LIN {X 0,Y 524.503,Z 419.032,A -85,B 0,C 180,E1 -2304.785,E2 -2304.785} C_VEL
LIN {X 0,Y 515.233,Z 402.102,A -85,B 0,C 180,E1 -2307.484,E2 -2307.484} C_VEL
LIN {X 0,Y 507.271,Z 387.982,A -85,B 0,C 180,E1 -2309.916,E2 -2309.916} C_VEL
LIN {X 0,Y 504.406,Z 383.021,A -85,B 0,C 180,E1 -2310.815,E2 -2310.815} C_VEL
LIN {X 0,Y 501.74,Z 378.349,A -85,B 0,C 180,E1 -2311.688,E2 -2311.688} C_VEL
LIN {X 0,Y 499.768,Z 374.769,A -85,B 0,C 180,E1 -2312.345,E2 -2312.345} C_VEL
LIN {X 0,Y 499.108,Z 373.613,A -85,B 0,C 180,E1 -2312.564,E2 -2312.564} C_VEL
LIN {X 0,Y 497.066,Z 370.383,A -85,B 0,C 180,E1 -2313.219,E2 -2313.219} C_VEL
LIN {X 0,Y 496.734,Z 368.862,A -85,B 0,C 180,E1 -2313.458,E2 -2313.458} C_VEL
LIN {X 0,Y 496.771,Z 368.854,A -85,B 0,C 180,E1 -2317.017,E2 -2317.017} C_VEL
LIN {X 0,Y 496.751,Z 368.855,A -85,B 0,C 180,E1 -2320.481,E2 -2320.481} C_VEL
LIN {X 0,Y 496.763,Z 368.853,A -85,B 0,C 180,E1 -2323.994,E2 -2323.994} C_VEL
LIN {X 0,Y 496.722,Z 368.861,A -85,B 0,C 180,E1 -2327.562,E2 -2327.562} C_VEL
LIN {X 0,Y 496.757,Z 368.858,A -85,B 0,C 180,E1 -2331.214,E2 -2331.214} C_VEL
LIN {X 0,Y 496.754,Z 368.857,A -85,B 0,C 180,E1 -2334.688,E2 -2334.688} C_VEL
LIN {X 0,Y 496.767,Z 368.858,A -85,B 0,C 180,E1 -2338.27,E2 -2338.27} C_VEL
LIN {X 0,Y 496.741,Z 368.864,A -85,B 0,C 180,E1 -2341.73,E2 -2341.73} C_VEL
LIN {X 0,Y 496.762,Z 368.856,A -85,B 0,C 180,E1 -2345.313,E2 -2345.313} C_VEL
LIN {X 0,Y 496.739,Z 368.861,A -85,B 0,C 180,E1 -2348.772,E2 -2348.772} C_VEL
LIN {X 0,Y 496.743,Z 368.861,A -85,B 0,C 180,E1 -2352.438,E2 -2352.438} C_VEL
LIN {X 0,Y 496.77,Z 368.855,A -85,B 0,C 180,E1 -2355.887,E2 -2355.887} C_VEL
LIN {X 0,Y 496.771,Z 368.857,A -85,B 0,C 180,E1 -2359.519,E2 -2359.519} C_VEL
LIN {X 0,Y 496.746,Z 368.856,A -85,B 0,C 180,E1 -2363.095,E2 -2363.095} C_VEL
LIN {X 0,Y 496.729,Z 368.857,A -85,B 0,C 180,E1 -2366.801,E2 -2366.801} C_VEL
LIN {X 0,Y 496.772,Z 368.856,A -85,B 0,C 180,E1 -2370.344,E2 -2370.344} C_VEL
LIN {X 0,Y 496.768,Z 368.854,A -85,B 0,C 180,E1 -2373.979,E2 -2373.979} C_VEL
LIN {X 0,Y 496.751,Z 368.842,A -85,B 0,C 180,E1 -2377.53,E2 -2377.53} C_VEL
LIN {X 0,Y 496.721,Z 368.855,A -85,B 0,C 180,E1 -2381.012,E2 -2381.012} C_VEL
LIN {X 0,Y 496.77,Z 368.857,A -85,B 0,C 180,E1 -2384.462,E2 -2384.462} C_VEL
LIN {X 0,Y 496.726,Z 368.853,A -85,B 0,C 180,E1 -2387.967,E2 -2387.967} C_VEL
LIN {X 0,Y 496.762,Z 368.844,A -85,B 0,C 180,E1 -2391.542,E2 -2391.542} C_VEL
LIN {X 0,Y 496.76,Z 368.858,A -85,B 0,C 180,E1 -2392.469,E2 -2392.469} C_VEL
LIN {X 0,Y 496.68,Z 369.647,A -85,B 0,C 180,E1 -2392.956,E2 -2392.956} C_VEL
LIN {X 0,Y 496.43,Z 372.237,A -85,B 0,C 180,E1 -2393.507,E2 -2393.507} C_VEL
LIN {X 0,Y 496.098,Z 377.593,A -85,B 0,C 180,E1 -2394.159,E2 -2394.159} C_VEL
LIN {X 0,Y 496.835,Z 388.981,A -85,B 0,C 180,E1 -2395.158,E2 -2395.158} C_VEL
LIN {X 0,Y 497.729,Z 392.512,A -85,B 0,C 180,E1 -2395.508,E2 -2395.508} C_VEL
LIN {X 0,Y 500.484,Z 400.044,A -85,B 0,C 180,E1 -2396.325,E2 -2396.325} C_VEL
LIN {X 0,Y 498.752,Z 444.32,A -85,B 0,C 180,E1 -2399.73,E2 -2399.73} C_VEL
LIN {X 0,Y 497.933,Z 478.056,A -85,B 0,C 180,E1 -2402.169,E2 -2402.169} C_VEL
LIN {X 0,Y 498.047,Z 482.397,A -85,B 0,C 180,E1 -2402.43,E2 -2402.43} C_VEL
LIN {X 0,Y 499.111,Z 490.744,A -85,B 0,C 180,E1 -2402.631,E2 -2402.631} C_VEL
LIN {X 0,Y 496.753,Z 690.079,A -85,B 0,C 180,E1 -2405.69,E2 -2405.69} C_VEL
LIN {X 0,Y 496.386,Z 708.436,A -85,B 0,C 180,E1 -2406.179,E2 -2406.179} C_VEL
LIN {X 0,Y 495.792,Z 726.382,A -85,B 0,C 180,E1 -2406.87,E2 -2406.87} C_VEL
LIN {X 0,Y 495,Z 743.469,A -85,B 0,C 180,E1 -2407.745,E2 -2407.745} C_VEL
LIN {X 0,Y 494.076,Z 760.052,A -85,B 0,C 180,E1 -2408.825,E2 -2408.825} C_VEL
LIN {X 0,Y 493.114,Z 775.645,A -85,B 0,C 180,E1 -2410.084,E2 -2410.084} C_VEL
LIN {X 0,Y 492.093,Z 790.238,A -85,B 0,C 180,E1 -2411.521,E2 -2411.521} C_VEL
LIN {X 0,Y 491.127,Z 803.548,A -85,B 0,C 180,E1 -2413.108,E2 -2413.108} C_VEL
LIN {X 0,Y 490.234,Z 815.743,A -85,B 0,C 180,E1 -2414.867,E2 -2414.867} C_VEL
LIN {X 0,Y 489.489,Z 826.599,A -85,B 0,C 180,E1 -2416.775,E2 -2416.775} C_VEL
LIN {X 0,Y 488.925,Z 835.924,A -85,B 0,C 180,E1 -2418.798,E2 -2418.798} C_VEL
LIN {X 0,Y 488.507,Z 843.713,A -85,B 0,C 180,E1 -2420.933,E2 -2420.933} C_VEL
LIN {X 0,Y 488.27,Z 849.911,A -85,B 0,C 180,E1 -2423.179,E2 -2423.179} C_VEL
LIN {X 0,Y 488.161,Z 854.237,A -85,B 0,C 180,E1 -2425.419,E2 -2425.419} C_VEL
LIN {X 0,Y 488.097,Z 856.834,A -85,B 0,C 180,E1 -2427.652,E2 -2427.652} C_VEL
LIN {X 0,Y 488.082,Z 857.774,A -85,B 0,C 180,E1 -2429.883,E2 -2429.883} C_VEL
LIN {X 0,Y 488.098,Z 857.016,A -85,B 0,C 180,E1 -2432.231,E2 -2432.231} C_VEL
LIN {X 0,Y 488.156,Z 854.577,A -85,B 0,C 180,E1 -2434.464,E2 -2434.464} C_VEL
LIN {X 0,Y 488.255,Z 850.404,A -85,B 0,C 180,E1 -2436.704,E2 -2436.704} C_VEL
LIN {X 0,Y 488.47,Z 844.75,A -85,B 0,C 180,E1 -2438.831,E2 -2438.831} C_VEL
LIN {X 0,Y 488.848,Z 837.248,A -85,B 0,C 180,E1 -2440.966,E2 -2440.966} C_VEL
LIN {X 0,Y 489.381,Z 828.236,A -85,B 0,C 180,E1 -2442.988,E2 -2442.988} C_VEL
LIN {X 0,Y 490.084,Z 817.732,A -85,B 0,C 180,E1 -2444.896,E2 -2444.896} C_VEL
LIN {X 0,Y 490.962,Z 805.709,A -85,B 0,C 180,E1 -2446.688,E2 -2446.688} C_VEL
LIN {X 0,Y 491.866,Z 793.128,A -85,B 0,C 180,E1 -2448.243,E2 -2448.243} C_VEL
LIN {X 0,Y 492.899,Z 778.54,A -85,B 0,C 180,E1 -2449.739,E2 -2449.739} C_VEL
LIN {X 0,Y 493.905,Z 762.904,A -85,B 0,C 180,E1 -2451.052,E2 -2451.052} C_VEL
LIN {X 0,Y 494.82,Z 746.936,A -85,B 0,C 180,E1 -2452.139,E2 -2452.139} C_VEL
LIN {X 0,Y 495.663,Z 729.626,A -85,B 0,C 180,E1 -2453.072,E2 -2453.072} C_VEL
LIN {X 0,Y 496.319,Z 711.178,A -85,B 0,C 180,E1 -2453.824,E2 -2453.824} C_VEL
LIN {X 0,Y 496.741,Z 692.317,A -85,B 0,C 180,E1 -2454.355,E2 -2454.355} C_VEL
LIN {X 0,Y 497.123,Z 656.576,A -85,B 0,C 180,E1 -2454.939,E2 -2454.939} C_VEL
LIN {X 0,Y 498.961,Z 488.001,A -85,B 0,C 180,E1 -2457.512,E2 -2457.512} C_VEL
LIN {X 0,Y 497.92,Z 481.292,A -85,B 0,C 180,E1 -2457.702,E2 -2457.702} C_VEL
LIN {X 0,Y 498.595,Z 448.895,A -85,B 0,C 180,E1 -2460.016,E2 -2460.016} C_VEL
LIN {X 0,Y 500.418,Z 403.002,A -85,B 0,C 180,E1 -2463.543,E2 -2463.543} C_VEL
LIN {X 0,Y 500.438,Z 400,A -85,B 0,C 180,E1 -2463.782,E2 -2463.782} C_VEL
LIN {X 0,Y 492.568,Z 379.479,A -85,B 0,C 180,E1 -2466.01,E2 -2466.01} C_VEL
LIN {X 0,Y 488.944,Z 370.528,A -85,B 0,C 180,E1 -2466.986,E2 -2466.986} C_VEL
LIN {X 0,Y 488.829,Z 369.846,A -85,B 0,C 180,E1 -2467.087,E2 -2467.087} C_VEL
LIN {X 0,Y 488.778,Z 369.84,A -85,B 0,C 180,E1 -2470.449,E2 -2470.449} C_VEL
LIN {X 0,Y 488.775,Z 369.837,A -85,B 0,C 180,E1 -2474.108,E2 -2474.108} C_VEL
LIN {X 0,Y 488.822,Z 369.832,A -85,B 0,C 180,E1 -2477.596,E2 -2477.596} C_VEL
LIN {X 0,Y 488.839,Z 370.058,A -85,B 0,C 180,E1 -2479.814,E2 -2479.814} C_VEL
LIN {X 0,Y 491.722,Z 377.094,A -85,B 0,C 180,E1 -2480.78,E2 -2480.78} C_VEL
LIN {X 0,Y 500.109,Z 397.524,A -85,B 0,C 180,E1 -2483.487,E2 -2483.487} C_VEL
LIN {X 0,Y 502.886,Z 405.19,A -85,B 0,C 180,E1 -2484.432,E2 -2484.432} C_VEL
LIN {X 0,Y 500.766,Z 444.723,A -85,B 0,C 180,E1 -2487.784,E2 -2487.784} C_VEL
LIN {X 0,Y 498.572,Z 486.822,A -85,B 0,C 180,E1 -2491.294,E2 -2491.294} C_VEL
LIN {X 0,Y 496.468,Z 530.886,A -85,B 0,C 180,E1 -2494.916,E2 -2494.916} C_VEL
LIN {X 0,Y 494.54,Z 576.296,A -85,B 0,C 180,E1 -2498.596,E2 -2498.596} C_VEL
LIN {X 0,Y 493.937,Z 594.847,A -85,B 0,C 180,E1 -2500.054,E2 -2500.054} C_VEL
LIN {X 0,Y 494.638,Z 602.56,A -85,B 0,C 180,E1 -2500.224,E2 -2500.224} C_VEL
LIN {X 0,Y 492.622,Z 739.25,A -85,B 0,C 180,E1 -2502.545,E2 -2502.545} C_VEL
LIN {X 0,Y 492.328,Z 756.165,A -85,B 0,C 180,E1 -2503.063,E2 -2503.063} C_VEL
LIN {X 0,Y 491.898,Z 771.737,A -85,B 0,C 180,E1 -2503.77,E2 -2503.77} C_VEL
LIN {X 0,Y 491.359,Z 786.911,A -85,B 0,C 180,E1 -2504.697,E2 -2504.697} C_VEL
LIN {X 0,Y 490.769,Z 800.72,A -85,B 0,C 180,E1 -2505.788,E2 -2505.788} C_VEL
LIN {X 0,Y 490.179,Z 813.819,A -85,B 0,C 180,E1 -2507.093,E2 -2507.093} C_VEL
LIN {X 0,Y 489.668,Z 824.783,A -85,B 0,C 180,E1 -2508.456,E2 -2508.456} C_VEL
LIN {X 0,Y 489.189,Z 835.467,A -85,B 0,C 180,E1 -2510.121,E2 -2510.121} C_VEL
LIN {X 0,Y 488.851,Z 843.777,A -85,B 0,C 180,E1 -2511.768,E2 -2511.768} C_VEL
LIN {X 0,Y 488.601,Z 851.044,A -85,B 0,C 180,E1 -2513.655,E2 -2513.655} C_VEL
LIN {X 0,Y 488.455,Z 856.104,A -85,B 0,C 180,E1 -2515.478,E2 -2515.478} C_VEL
LIN {X 0,Y 488.405,Z 859.682,A -85,B 0,C 180,E1 -2517.484,E2 -2517.484} C_VEL
LIN {X 0,Y 488.391,Z 861.302,A -85,B 0,C 180,E1 -2519.413,E2 -2519.413} C_VEL
LIN {X 0,Y 488.438,Z 861.141,A -85,B 0,C 180,E1 -2521.407,E2 -2521.407} C_VEL
LIN {X 0,Y 488.505,Z 859.288,A -85,B 0,C 180,E1 -2523.285,E2 -2523.285} C_VEL
LIN {X 0,Y 488.672,Z 855.426,A -85,B 0,C 180,E1 -2525.283,E2 -2525.283} C_VEL
LIN {X 0,Y 488.903,Z 850.255,A -85,B 0,C 180,E1 -2527.048,E2 -2527.048} C_VEL
LIN {X 0,Y 489.295,Z 842.689,A -85,B 0,C 180,E1 -2528.934,E2 -2528.934} C_VEL
LIN {X 0,Y 489.739,Z 833.97,A -85,B 0,C 180,E1 -2530.588,E2 -2530.588} C_VEL
LIN {X 0,Y 490.294,Z 823.742,A -85,B 0,C 180,E1 -2532.125,E2 -2532.125} C_VEL
LIN {X 0,Y 490.912,Z 812.346,A -85,B 0,C 180,E1 -2533.486,E2 -2533.486} C_VEL
LIN {X 0,Y 491.551,Z 799.331,A -85,B 0,C 180,E1 -2534.729,E2 -2534.729} C_VEL
LIN {X 0,Y 492.105,Z 785.893,A -85,B 0,C 180,E1 -2535.738,E2 -2535.738} C_VEL
LIN {X 0,Y 492.623,Z 770.434,A -85,B 0,C 180,E1 -2536.629,E2 -2536.629} C_VEL
LIN {X 0,Y 492.938,Z 754.963,A -85,B 0,C 180,E1 -2537.271,E2 -2537.271} C_VEL
LIN {X 0,Y 493.11,Z 738.497,A -85,B 0,C 180,E1 -2537.722,E2 -2537.722} C_VEL
LIN {X 0,Y 495.144,Z 663.885,A -85,B 0,C 180,E1 -2539.24,E2 -2539.24} C_VEL
LIN {X 0,Y 497.519,Z 607.496,A -85,B 0,C 180,E1 -2540.468,E2 -2540.468} C_VEL
LIN {X 0,Y 498.963,Z 602.16,A -85,B 0,C 180,E1 -2540.835,E2 -2540.835} C_VEL
LIN {X 0,Y 502.913,Z 561.509,A -85,B 0,C 180,E1 -2544.489,E2 -2544.489} C_VEL
LIN {X 0,Y 508.091,Z 522.478,A -85,B 0,C 180,E1 -2548.183,E2 -2548.183} C_VEL
LIN {X 0,Y 513.352,Z 494.26,A -85,B 0,C 180,E1 -2551.019,E2 -2551.019} C_VEL
LIN {X 0,Y 519.178,Z 471.939,A -85,B 0,C 180,E1 -2553.421,E2 -2553.421} C_VEL
LIN {X 0,Y 525.35,Z 455.383,A -85,B 0,C 180,E1 -2555.35,E2 -2555.35} C_VEL
LIN {X 0,Y 527.979,Z 449.901,A -85,B 0,C 180,E1 -2556.037,E2 -2556.037} C_VEL
LIN {X 0,Y 520.798,Z 461.366,A -85,B 0,C 180,E1 -2557.27,E2 -2557.27} C_VEL
LIN {X 0,Y 516.041,Z 472.438,A -85,B 0,C 180,E1 -2558.484,E2 -2558.484} C_VEL
LIN {X 0,Y 513.414,Z 483.465,A -85,B 0,C 180,E1 -2559.713,E2 -2559.713} C_VEL
LIN {X 0,Y 512.933,Z 495.108,A -85,B 0,C 180,E1 -2561.028,E2 -2561.028} C_VEL
LIN {X 0,Y 514.549,Z 505.694,A -85,B 0,C 180,E1 -2562.247,E2 -2562.247} C_VEL
LIN {X 0,Y 518.036,Z 515.468,A -85,B 0,C 180,E1 -2563.402,E2 -2563.402} C_VEL
LIN {X 0,Y 523.717,Z 525.213,A -85,B 0,C 180,E1 -2564.592,E2 -2564.592} C_VEL
LIN {X 0,Y 531.685,Z 534.476,A -85,B 0,C 180,E1 -2565.765,E2 -2565.765} C_VEL
LIN {X 0,Y 541.467,Z 542.475,A -85,B 0,C 180,E1 -2566.835,E2 -2566.835} C_VEL
LIN {X 0,Y 552.276,Z 548.88,A -85,B 0,C 180,E1 -2567.771,E2 -2567.771} C_VEL
LIN {X 0,Y 562.809,Z 553.266,A -85,B 0,C 180,E1 -2568.564,E2 -2568.564} C_VEL
LIN {X 0,Y 567.662,Z 554.303,A -85,B 0,C 180,E1 -2569.08,E2 -2569.08} C_VEL
LIN {X 0,Y 570.982,Z 554.208,A -85,B 0,C 180,E1 -2569.617,E2 -2569.617} C_VEL
LIN {X 0,Y 573.098,Z 553.255,A -85,B 0,C 180,E1 -2570.186,E2 -2570.186} C_VEL
LIN {X 0,Y 573.653,Z 552.573,A -85,B 0,C 180,E1 -2570.46,E2 -2570.46} C_VEL
LIN {X 0,Y 566.628,Z 573.364,A -85,B 0,C 180,E1 -2570.751,E2 -2570.751} C_VEL
LIN {X 0,Y 562.375,Z 585.951,A -85,B 0,C 180,E1 -2571.06,E2 -2571.06} C_VEL
LIN {X 0,Y 553.254,Z 606.117,A -85,B 0,C 180,E1 -2571.202,E2 -2571.202} C_VEL
LIN {X 0,Y 542.151,Z 627.242,A -85,B 0,C 180,E1 -2571.506,E2 -2571.506} C_VEL
LIN {X 0,Y 532.299,Z 645.678,A -85,B 0,C 180,E1 -2571.967,E2 -2571.967} C_VEL
LIN {X 0,Y 525.341,Z 661.055,A -85,B 0,C 180,E1 -2572.479,E2 -2572.479} C_VEL
LIN {X 0,Y 521.674,Z 671.361,A -85,B 0,C 180,E1 -2572.874,E2 -2572.874} C_VEL
LIN {X 0,Y 515.253,Z 685.606,A -85,B 0,C 180,E1 -2573.365,E2 -2573.365} C_VEL
LIN {X 0,Y 507.043,Z 711.323,A -85,B 0,C 180,E1 -2574.428,E2 -2574.428} C_VEL
LIN {X 0,Y 504.91,Z 720.444,A -85,B 0,C 180,E1 -2574.812,E2 -2574.812} C_VEL
LIN {X 0,Y 504.327,Z 762.509,A -85,B 0,C 180,E1 -2575.46,E2 -2575.46} C_VEL
LIN {X 0,Y 503.48,Z 786.582,A -85,B 0,C 180,E1 -2576.043,E2 -2576.043} C_VEL
LIN {X 0,Y 502.543,Z 808.772,A -85,B 0,C 180,E1 -2576.794,E2 -2576.794} C_VEL
LIN {X 0,Y 501.448,Z 827.405,A -85,B 0,C 180,E1 -2577.63,E2 -2577.63} C_VEL
LIN {X 0,Y 499.915,Z 846.819,A -85,B 0,C 180,E1 -2578.733,E2 -2578.733} C_VEL
LIN {X 0,Y 498.233,Z 866.627,A -85,B 0,C 180,E1 -2580.104,E2 -2580.104} C_VEL
LIN {X 0,Y 496.476,Z 885.398,A -85,B 0,C 180,E1 -2581.651,E2 -2581.651} C_VEL
LIN {X 0,Y 494.727,Z 904.088,A -85,B 0,C 180,E1 -2583.471,E2 -2583.471} C_VEL
LIN {X 0,Y 493.156,Z 920.729,A -85,B 0,C 180,E1 -2585.377,E2 -2585.377} C_VEL
LIN {X 0,Y 491.772,Z 935.909,A -85,B 0,C 180,E1 -2587.401,E2 -2587.401} C_VEL
LIN {X 0,Y 490.566,Z 950.305,A -85,B 0,C 180,E1 -2589.645,E2 -2589.645} C_VEL
LIN {X 0,Y 489.601,Z 963.337,A -85,B 0,C 180,E1 -2592.039,E2 -2592.039} C_VEL
LIN {X 0,Y 488.902,Z 974.404,A -85,B 0,C 180,E1 -2594.46,E2 -2594.46} C_VEL
LIN {X 0,Y 488.404,Z 984.338,A -85,B 0,C 180,E1 -2597.106,E2 -2597.106} C_VEL
LIN {X 0,Y 488.115,Z 992.2,A -85,B 0,C 180,E1 -2599.734,E2 -2599.734} C_VEL
LIN {X 0,Y 487.964,Z 998.151,A -85,B 0,C 180,E1 -2602.346,E2 -2602.346} C_VEL
LIN {X 0,Y 487.907,Z 1002.147,A -85,B 0,C 180,E1 -2604.838,E2 -2604.838} C_VEL
LIN {X 0,Y 487.895,Z 1004.524,A -85,B 0,C 180,E1 -2607.298,E2 -2607.298} C_VEL
LIN {X 0,Y 487.897,Z 1005.44,A -85,B 0,C 180,E1 -2609.647,E2 -2609.647} C_VEL
LIN {X 0,Y 487.91,Z 1004.912,A -85,B 0,C 180,E1 -2612.114,E2 -2612.114} C_VEL
LIN {X 0,Y 487.912,Z 1002.74,A -85,B 0,C 180,E1 -2614.702,E2 -2614.702} C_VEL
LIN {X 0,Y 487.947,Z 998.808,A -85,B 0,C 180,E1 -2617.299,E2 -2617.299} C_VEL
LIN {X 0,Y 488.067,Z 993.353,A -85,B 0,C 180,E1 -2619.811,E2 -2619.811} C_VEL
LIN {X 0,Y 488.311,Z 986.309,A -85,B 0,C 180,E1 -2622.295,E2 -2622.295} C_VEL
LIN {X 0,Y 488.737,Z 977.337,A -85,B 0,C 180,E1 -2624.816,E2 -2624.816} C_VEL
LIN {X 0,Y 489.401,Z 966.295,A -85,B 0,C 180,E1 -2627.354,E2 -2627.354} C_VEL
LIN {X 0,Y 490.31,Z 953.621,A -85,B 0,C 180,E1 -2629.786,E2 -2629.786} C_VEL
LIN {X 0,Y 491.493,Z 939.294,A -85,B 0,C 180,E1 -2632.108,E2 -2632.108} C_VEL
LIN {X 0,Y 492.935,Z 923.225,A -85,B 0,C 180,E1 -2634.315,E2 -2634.315} C_VEL
LIN {X 0,Y 494.614,Z 905.274,A -85,B 0,C 180,E1 -2636.406,E2 -2636.406} C_VEL
LIN {X 0,Y 496.38,Z 886.455,A -85,B 0,C 180,E1 -2638.252,E2 -2638.252} C_VEL
LIN {X 0,Y 498.176,Z 867.207,A -85,B 0,C 180,E1 -2639.851,E2 -2639.851} C_VEL
LIN {X 0,Y 499.838,Z 847.827,A -85,B 0,C 180,E1 -2641.204,E2 -2641.204} C_VEL
LIN {X 0,Y 501.365,Z 828.672,A -85,B 0,C 180,E1 -2642.307,E2 -2642.307} C_VEL
LIN {X 0,Y 502.601,Z 808.206,A -85,B 0,C 180,E1 -2643.234,E2 -2643.234} C_VEL
LIN {X 0,Y 503.712,Z 785.487,A -85,B 0,C 180,E1 -2644.029,E2 -2644.029} C_VEL
LIN {X 0,Y 504.625,Z 762.44,A -85,B 0,C 180,E1 -2644.609,E2 -2644.609} C_VEL
LIN {X 0,Y 505.297,Z 722.062,A -85,B 0,C 180,E1 -2645.262,E2 -2645.262} C_VEL
LIN {X 0,Y 505.606,Z 719.266,A -85,B 0,C 180,E1 -2645.34,E2 -2645.34} C_VEL
LIN {X 0,Y 509.96,Z 703.556,A -85,B 0,C 180,E1 -2646.029,E2 -2646.029} C_VEL
LIN {X 0,Y 516.417,Z 684.139,A -85,B 0,C 180,E1 -2646.795,E2 -2646.795} C_VEL
LIN {X 0,Y 522.774,Z 669.701,A -85,B 0,C 180,E1 -2647.253,E2 -2647.253} C_VEL
LIN {X 0,Y 527.202,Z 657.309,A -85,B 0,C 180,E1 -2647.707,E2 -2647.707} C_VEL
LIN {X 0,Y 535.529,Z 639.572,A -85,B 0,C 180,E1 -2648.214,E2 -2648.214} C_VEL
LIN {X 0,Y 546.551,Z 619.139,A -85,B 0,C 180,E1 -2648.634,E2 -2648.634} C_VEL
LIN {X 0,Y 556.954,Z 598.362,A -85,B 0,C 180,E1 -2648.867,E2 -2648.867} C_VEL
LIN {X 0,Y 562.84,Z 584.646,A -85,B 0,C 180,E1 -2648.966,E2 -2648.966} C_VEL
LIN {X 0,Y 567.532,Z 570.757,A -85,B 0,C 180,E1 -2649.298,E2 -2649.298} C_VEL
LIN {X 0,Y 573.649,Z 552.565,A -85,B 0,C 180,E1 -2649.551,E2 -2649.551} C_VEL
LIN {X 0,Y 571.887,Z 553.958,A -85,B 0,C 180,E1 -2650.18,E2 -2650.18} C_VEL
LIN {X 0,Y 568.861,Z 554.372,A -85,B 0,C 180,E1 -2650.752,E2 -2650.752} C_VEL
LIN {X 0,Y 565.013,Z 553.856,A -85,B 0,C 180,E1 -2651.229,E2 -2651.229} C_VEL
LIN {X 0,Y 554.055,Z 550.104,A -85,B 0,C 180,E1 -2652.308,E2 -2652.308} C_VEL
LIN {X 0,Y 544.18,Z 544.7,A -85,B 0,C 180,E1 -2653.468,E2 -2653.468} C_VEL
LIN {X 0,Y 535.663,Z 537.821,A -85,B 0,C 180,E1 -2654.67,E2 -2654.67} C_VEL
LIN {X 0,Y 528.131,Z 528.834,A -85,B 0,C 180,E1 -2655.989,E2 -2655.989} C_VEL
LIN {X 0,Y 522.652,Z 519.047,A -85,B 0,C 180,E1 -2657.225,E2 -2657.225} C_VEL
LIN {X 0,Y 518.636,Z 507.922,A -85,B 0,C 180,E1 -2658.457,E2 -2658.457} C_VEL
LIN {X 0,Y 516.125,Z 495.378,A -85,B 0,C 180,E1 -2659.682,E2 -2659.682} C_VEL
LIN {X 0,Y 514.966,Z 479.928,A -85,B 0,C 180,E1 -2661.018,E2 -2661.018} C_VEL
LIN {X 0,Y 515.59,Z 460.544,A -85,B 0,C 180,E1 -2662.489,E2 -2662.489} C_VEL
LIN {X 0,Y 518.516,Z 423.387,A -85,B 0,C 180,E1 -2665.196,E2 -2665.196} C_VEL
LIN {X 0,Y 509.071,Z 406.235,A -85,B 0,C 180,E1 -2667.974,E2 -2667.974} C_VEL
LIN {X 0,Y 502.092,Z 393.774,A -85,B 0,C 180,E1 -2670.143,E2 -2670.143} C_VEL
LIN {X 0,Y 496.676,Z 384.303,A -85,B 0,C 180,E1 -2671.897,E2 -2671.897} C_VEL
LIN {X 0,Y 494.04,Z 379.628,A -85,B 0,C 180,E1 -2672.782,E2 -2672.782} C_VEL
LIN {X 0,Y 492.051,Z 376.345,A -85,B 0,C 180,E1 -2673.446,E2 -2673.446} C_VEL
LIN {X 0,Y 491.125,Z 374.539,A -85,B 0,C 180,E1 -2673.783,E2 -2673.783} C_VEL
LIN {X 0,Y 489.128,Z 371.287,A -85,B 0,C 180,E1 -2674.449,E2 -2674.449} C_VEL
LIN {X 0,Y 488.803,Z 369.847,A -85,B 0,C 180,E1 -2674.705,E2 -2674.705} C_VEL
LIN {X 0,Y 488.835,Z 369.843,A -85,B 0,C 180,E1 -2678.271,E2 -2678.271} C_VEL
LIN {X 0,Y 488.828,Z 369.843,A -85,B 0,C 180,E1 -2682.011,E2 -2682.011} C_VEL
LIN {X 0,Y 488.809,Z 369.847,A -85,B 0,C 180,E1 -2685.549,E2 -2685.549} C_VEL
LIN {X 0,Y 488.796,Z 369.849,A -85,B 0,C 180,E1 -2689.153,E2 -2689.153} C_VEL
LIN {X 0,Y 488.828,Z 369.844,A -85,B 0,C 180,E1 -2692.597,E2 -2692.597} C_VEL
LIN {X 0,Y 488.798,Z 369.849,A -85,B 0,C 180,E1 -2696.247,E2 -2696.247} C_VEL
LIN {X 0,Y 488.832,Z 369.85,A -85,B 0,C 180,E1 -2699.766,E2 -2699.766} C_VEL
LIN {X 0,Y 488.81,Z 369.851,A -85,B 0,C 180,E1 -2703.284,E2 -2703.284} C_VEL
LIN {X 0,Y 488.823,Z 369.848,A -85,B 0,C 180,E1 -2706.814,E2 -2706.814} C_VEL
LIN {X 0,Y 488.781,Z 369.848,A -85,B 0,C 180,E1 -2710.371,E2 -2710.371} C_VEL
LIN {X 0,Y 488.821,Z 369.846,A -85,B 0,C 180,E1 -2713.967,E2 -2713.967} C_VEL
LIN {X 0,Y 488.818,Z 369.848,A -85,B 0,C 180,E1 -2717.499,E2 -2717.499} C_VEL
LIN {X 0,Y 488.829,Z 369.844,A -85,B 0,C 180,E1 -2721.1,E2 -2721.1} C_VEL
LIN {X 0,Y 488.789,Z 369.849,A -85,B 0,C 180,E1 -2724.665,E2 -2724.665} C_VEL
LIN {X 0,Y 488.816,Z 369.842,A -85,B 0,C 180,E1 -2728.33,E2 -2728.33} C_VEL
LIN {X 0,Y 488.805,Z 369.84,A -85,B 0,C 180,E1 -2731.716,E2 -2731.716} C_VEL
LIN {X 0,Y 488.812,Z 369.831,A -85,B 0,C 180,E1 -2735.299,E2 -2735.299} C_VEL
LIN {X 0,Y 488.826,Z 369.843,A -85,B 0,C 180,E1 -2738.803,E2 -2738.803} C_VEL
LIN {X 0,Y 488.824,Z 369.826,A -85,B 0,C 180,E1 -2742.454,E2 -2742.454} C_VEL
LIN {X 0,Y 488.804,Z 369.845,A -85,B 0,C 180,E1 -2745.935,E2 -2745.935} C_VEL
LIN {X 0,Y 488.795,Z 369.854,A -85,B 0,C 180,E1 -2749.576,E2 -2749.576} C_VEL
LIN {X 0,Y 488.855,Z 370.012,A -85,B 0,C 180,E1 -2753.062,E2 -2753.062} C_VEL
LIN {X 0,Y 497.729,Z 392.512,A -85,B 0,C 180,E1 -2755.508,E2 -2755.508} C_VEL
LIN {X 0,Y 498.073,Z 395.994,A -85,B 0,C 180,E1 -2755.811,E2 -2755.811} C_VEL
LIN {X 0,Y 496.56,Z 401.823,A -85,B 0,C 180,E1 -2756.156,E2 -2756.156} C_VEL
LIN {X 0,Y 493.439,Z 410.585,A -85,B 0,C 180,E1 -2756.62,E2 -2756.62} C_VEL
LIN {X 0,Y 493.054,Z 413.215,A -85,B 0,C 180,E1 -2756.804,E2 -2756.804} C_VEL
LIN {X 0,Y 491.393,Z 456.207,A -85,B 0,C 180,E1 -2760.099,E2 -2760.099} C_VEL
LIN {X 0,Y 490.934,Z 483.139,A -85,B 0,C 180,E1 -2761.989,E2 -2761.989} C_VEL
LIN {X 0,Y 492.064,Z 491.769,A -85,B 0,C 180,E1 -2762.204,E2 -2762.204} C_VEL
LIN {X 0,Y 489.525,Z 691.201,A -85,B 0,C 180,E1 -2765.307,E2 -2765.307} C_VEL
LIN {X 0,Y 489.144,Z 709.676,A -85,B 0,C 180,E1 -2765.805,E2 -2765.805} C_VEL
LIN {X 0,Y 488.522,Z 727.692,A -85,B 0,C 180,E1 -2766.51,E2 -2766.51} C_VEL
LIN {X 0,Y 487.691,Z 744.691,A -85,B 0,C 180,E1 -2767.393,E2 -2767.393} C_VEL
LIN {X 0,Y 486.71,Z 761.37,A -85,B 0,C 180,E1 -2768.495,E2 -2768.495} C_VEL
LIN {X 0,Y 485.688,Z 776.887,A -85,B 0,C 180,E1 -2769.767,E2 -2769.767} C_VEL
LIN {X 0,Y 484.595,Z 791.488,A -85,B 0,C 180,E1 -2771.224,E2 -2771.224} C_VEL
LIN {X 0,Y 483.576,Z 804.561,A -85,B 0,C 180,E1 -2772.803,E2 -2772.803} C_VEL
LIN {X 0,Y 482.592,Z 817.003,A -85,B 0,C 180,E1 -2774.622,E2 -2774.622} C_VEL
LIN {X 0,Y 481.778,Z 827.862,A -85,B 0,C 180,E1 -2776.56,E2 -2776.56} C_VEL
LIN {X 0,Y 481.153,Z 837.189,A -85,B 0,C 180,E1 -2778.615,E2 -2778.615} C_VEL
LIN {X 0,Y 480.685,Z 844.979,A -85,B 0,C 180,E1 -2780.784,E2 -2780.784} C_VEL
LIN {X 0,Y 480.411,Z 851.177,A -85,B 0,C 180,E1 -2783.067,E2 -2783.067} C_VEL
LIN {X 0,Y 480.278,Z 855.502,A -85,B 0,C 180,E1 -2785.343,E2 -2785.343} C_VEL
LIN {X 0,Y 480.202,Z 858.098,A -85,B 0,C 180,E1 -2787.614,E2 -2787.614} C_VEL
LIN {X 0,Y 480.183,Z 859.038,A -85,B 0,C 180,E1 -2789.881,E2 -2789.881} C_VEL
LIN {X 0,Y 480.202,Z 858.279,A -85,B 0,C 180,E1 -2792.268,E2 -2792.268} C_VEL
LIN {X 0,Y 480.273,Z 855.839,A -85,B 0,C 180,E1 -2794.538,E2 -2794.538} C_VEL
LIN {X 0,Y 480.394,Z 851.667,A -85,B 0,C 180,E1 -2796.814,E2 -2796.814} C_VEL
LIN {X 0,Y 480.642,Z 846.011,A -85,B 0,C 180,E1 -2798.976,E2 -2798.976} C_VEL
LIN {X 0,Y 481.068,Z 838.508,A -85,B 0,C 180,E1 -2801.145,E2 -2801.145} C_VEL
LIN {X 0,Y 481.659,Z 829.493,A -85,B 0,C 180,E1 -2803.2,E2 -2803.2} C_VEL
LIN {X 0,Y 482.429,Z 818.984,A -85,B 0,C 180,E1 -2805.138,E2 -2805.138} C_VEL
LIN {X 0,Y 483.379,Z 806.955,A -85,B 0,C 180,E1 -2806.957,E2 -2806.957} C_VEL
LIN {X 0,Y 484.397,Z 793.84,A -85,B 0,C 180,E1 -2808.597,E2 -2808.597} C_VEL
LIN {X 0,Y 485.495,Z 779.333,A -85,B 0,C 180,E1 -2810.096,E2 -2810.096} C_VEL
LIN {X 0,Y 486.566,Z 763.623,A -85,B 0,C 180,E1 -2811.426,E2 -2811.426} C_VEL
LIN {X 0,Y 487.562,Z 747.183,A -85,B 0,C 180,E1 -2812.55,E2 -2812.55} C_VEL
LIN {X 0,Y 488.462,Z 729.443,A -85,B 0,C 180,E1 -2813.503,E2 -2813.503} C_VEL
LIN {X 0,Y 489.112,Z 710.984,A -85,B 0,C 180,E1 -2814.243,E2 -2814.243} C_VEL
LIN {X 0,Y 489.518,Z 692.403,A -85,B 0,C 180,E1 -2814.758,E2 -2814.758} C_VEL
LIN {X 0,Y 490.104,Z 642.033,A -85,B 0,C 180,E1 -2815.57,E2 -2815.57} C_VEL
LIN {X 0,Y 491.911,Z 489.03,A -85,B 0,C 180,E1 -2817.942,E2 -2817.942} C_VEL
LIN {X 0,Y 490.878,Z 482.661,A -85,B 0,C 180,E1 -2818.119,E2 -2818.119} C_VEL
LIN {X 0,Y 491.556,Z 450.643,A -85,B 0,C 180,E1 -2820.407,E2 -2820.407} C_VEL
LIN {X 0,Y 493.432,Z 404.906,A -85,B 0,C 180,E1 -2823.936,E2 -2823.936} C_VEL
LIN {X 0,Y 493.32,Z 402.834,A -85,B 0,C 180,E1 -2824.111,E2 -2824.111} C_VEL
LIN {X 0,Y 485.048,Z 381.238,A -85,B 0,C 180,E1 -2826.492,E2 -2826.492} C_VEL
LIN {X 0,Y 480.904,Z 371.185,A -85,B 0,C 180,E1 -2827.613,E2 -2827.613} C_VEL
LIN {X 0,Y 480.849,Z 370.84,A -85,B 0,C 180,E1 -2827.686,E2 -2827.686} C_VEL
LIN {X 0,Y 480.899,Z 370.822,A -85,B 0,C 180,E1 -2831.179,E2 -2831.179} C_VEL
LIN {X 0,Y 480.842,Z 370.823,A -85,B 0,C 180,E1 -2834.671,E2 -2834.671} C_VEL
LIN {X 0,Y 480.837,Z 370.825,A -85,B 0,C 180,E1 -2838.29,E2 -2838.29} C_VEL
LIN {X 0,Y 480.888,Z 371.027,A -85,B 0,C 180,E1 -2839.084,E2 -2839.084} C_VEL
LIN {X 0,Y 490.099,Z 393.057,A -85,B 0,C 180,E1 -2842.142,E2 -2842.142} C_VEL
LIN {X 0,Y 496.011,Z 408.442,A -85,B 0,C 180,E1 -2844.116,E2 -2844.116} C_VEL
LIN {X 0,Y 493.608,Z 449.502,A -85,B 0,C 180,E1 -2847.638,E2 -2847.638} C_VEL
LIN {X 0,Y 491.327,Z 491.53,A -85,B 0,C 180,E1 -2851.164,E2 -2851.164} C_VEL
LIN {X 0,Y 489.044,Z 536.834,A -85,B 0,C 180,E1 -2854.922,E2 -2854.922} C_VEL
LIN {X 0,Y 486.925,Z 584.474,A -85,B 0,C 180,E1 -2858.813,E2 -2858.813} C_VEL
LIN {X 0,Y 486.56,Z 595.568,A -85,B 0,C 180,E1 -2859.683,E2 -2859.683} C_VEL
LIN {X 0,Y 487.281,Z 603.269,A -85,B 0,C 180,E1 -2859.864,E2 -2859.864} C_VEL
LIN {X 0,Y 485.047,Z 740.362,A -85,B 0,C 180,E1 -2862.261,E2 -2862.261} C_VEL
LIN {X 0,Y 484.734,Z 757.33,A -85,B 0,C 180,E1 -2862.793,E2 -2862.793} C_VEL
LIN {X 0,Y 484.281,Z 772.764,A -85,B 0,C 180,E1 -2863.507,E2 -2863.507} C_VEL
LIN {X 0,Y 483.699,Z 788.281,A -85,B 0,C 180,E1 -2864.473,E2 -2864.473} C_VEL
LIN {X 0,Y 483.084,Z 801.761,A -85,B 0,C 180,E1 -2865.557,E2 -2865.557} C_VEL
LIN {X 0,Y 482.477,Z 814.336,A -85,B 0,C 180,E1 -2866.823,E2 -2866.823} C_VEL
LIN {X 0,Y 481.902,Z 825.882,A -85,B 0,C 180,E1 -2868.268,E2 -2868.268} C_VEL
LIN {X 0,Y 481.385,Z 836.563,A -85,B 0,C 180,E1 -2869.952,E2 -2869.952} C_VEL
LIN {X 0,Y 481.014,Z 844.956,A -85,B 0,C 180,E1 -2871.633,E2 -2871.633} C_VEL
LIN {X 0,Y 480.739,Z 852.269,A -85,B 0,C 180,E1 -2873.551,E2 -2873.551} C_VEL
LIN {X 0,Y 480.583,Z 857.245,A -85,B 0,C 180,E1 -2875.346,E2 -2875.346} C_VEL
LIN {X 0,Y 480.521,Z 860.901,A -85,B 0,C 180,E1 -2877.376,E2 -2877.376} C_VEL
LIN {X 0,Y 480.508,Z 862.618,A -85,B 0,C 180,E1 -2879.284,E2 -2879.284} C_VEL
LIN {X 0,Y 480.556,Z 862.581,A -85,B 0,C 180,E1 -2881.311,E2 -2881.311} C_VEL
LIN {X 0,Y 480.641,Z 860.886,A -85,B 0,C 180,E1 -2883.219,E2 -2883.219} C_VEL
LIN {X 0,Y 480.82,Z 857.15,A -85,B 0,C 180,E1 -2885.249,E2 -2885.249} C_VEL
LIN {X 0,Y 481.082,Z 852.153,A -85,B 0,C 180,E1 -2887.043,E2 -2887.043} C_VEL
LIN {X 0,Y 481.464,Z 845.251,A -85,B 0,C 180,E1 -2888.84,E2 -2888.84} C_VEL
LIN {X 0,Y 481.956,Z 836.932,A -85,B 0,C 180,E1 -2890.519,E2 -2890.519} C_VEL
LIN {X 0,Y 482.525,Z 827.033,A -85,B 0,C 180,E1 -2892.08,E2 -2892.08} C_VEL
LIN {X 0,Y 483.204,Z 815.648,A -85,B 0,C 180,E1 -2893.522,E2 -2893.522} C_VEL
LIN {X 0,Y 483.875,Z 803.132,A -85,B 0,C 180,E1 -2894.779,E2 -2894.779} C_VEL
LIN {X 0,Y 484.522,Z 789.543,A -85,B 0,C 180,E1 -2895.868,E2 -2895.868} C_VEL
LIN {X 0,Y 485.042,Z 774.737,A -85,B 0,C 180,E1 -2896.773,E2 -2896.773} C_VEL
LIN {X 0,Y 485.439,Z 759.257,A -85,B 0,C 180,E1 -2897.477,E2 -2897.477} C_VEL
LIN {X 0,Y 485.626,Z 742.723,A -85,B 0,C 180,E1 -2897.973,E2 -2897.973} C_VEL
LIN {X 0,Y 487.821,Z 670.656,A -85,B 0,C 180,E1 -2899.533,E2 -2899.533} C_VEL
LIN {X 0,Y 490.82,Z 609.716,A -85,B 0,C 180,E1 -2900.947,E2 -2900.947} C_VEL
LIN {X 0,Y 492.502,Z 603.638,A -85,B 0,C 180,E1 -2901.371,E2 -2901.371} C_VEL
LIN {X 0,Y 497.184,Z 560.839,A -85,B 0,C 180,E1 -2905.299,E2 -2905.299} C_VEL
LIN {X 0,Y 502.752,Z 523.775,A -85,B 0,C 180,E1 -2908.899,E2 -2908.899} C_VEL
LIN {X 0,Y 508.269,Z 497.727,A -85,B 0,C 180,E1 -2911.592,E2 -2911.592} C_VEL
LIN {X 0,Y 514.093,Z 477.831,A -85,B 0,C 180,E1 -2913.796,E2 -2913.796} C_VEL
LIN {X 0,Y 520.513,Z 462.288,A -85,B 0,C 180,E1 -2915.654,E2 -2915.654} C_VEL
LIN {X 0,Y 521.646,Z 460.023,A -85,B 0,C 180,E1 -2915.968,E2 -2915.968} C_VEL
LIN {X 0,Y 514.762,Z 471.03,A -85,B 0,C 180,E1 -2917.214,E2 -2917.214} C_VEL
LIN {X 0,Y 510.208,Z 481.828,A -85,B 0,C 180,E1 -2918.472,E2 -2918.472} C_VEL
LIN {X 0,Y 507.95,Z 491.919,A -85,B 0,C 180,E1 -2919.677,E2 -2919.677} C_VEL
LIN {X 0,Y 507.649,Z 502.763,A -85,B 0,C 180,E1 -2920.985,E2 -2920.985} C_VEL
LIN {X 0,Y 509.591,Z 513.482,A -85,B 0,C 180,E1 -2922.298,E2 -2922.298} C_VEL
LIN {X 0,Y 513.205,Z 522.69,A -85,B 0,C 180,E1 -2923.451,E2 -2923.451} C_VEL
LIN {X 0,Y 518.563,Z 531.482,A -85,B 0,C 180,E1 -2924.574,E2 -2924.574} C_VEL
LIN {X 0,Y 526.289,Z 540.379,A -85,B 0,C 180,E1 -2925.744,E2 -2925.744} C_VEL
LIN {X 0,Y 535.951,Z 548.334,A -85,B 0,C 180,E1 -2926.839,E2 -2926.839} C_VEL
LIN {X 0,Y 547.472,Z 555.259,A -85,B 0,C 180,E1 -2927.858,E2 -2927.858} C_VEL
LIN {X 0,Y 559.715,Z 560.386,A -85,B 0,C 180,E1 -2928.769,E2 -2928.769} C_VEL
LIN {X 0,Y 564.758,Z 561.529,A -85,B 0,C 180,E1 -2929.265,E2 -2929.265} C_VEL
LIN {X 0,Y 568.232,Z 561.713,A -85,B 0,C 180,E1 -2929.798,E2 -2929.798} C_VEL
LIN {X 0,Y 561.005,Z 579.487,A -85,B 0,C 180,E1 -2930.154,E2 -2930.154} C_VEL
LIN {X 0,Y 558.539,Z 586.008,A -85,B 0,C 180,E1 -2930.332,E2 -2930.332} C_VEL
LIN {X 0,Y 547.964,Z 605.065,A -85,B 0,C 180,E1 -2930.58,E2 -2930.58} C_VEL
LIN {X 0,Y 533.173,Z 629.737,A -85,B 0,C 180,E1 -2931.149,E2 -2931.149} C_VEL
LIN {X 0,Y 522.892,Z 649.225,A -85,B 0,C 180,E1 -2931.717,E2 -2931.717} C_VEL
LIN {X 0,Y 516.784,Z 663.945,A -85,B 0,C 180,E1 -2932.24,E2 -2932.24} C_VEL
LIN {X 0,Y 514.597,Z 670.004,A -85,B 0,C 180,E1 -2932.473,E2 -2932.473} C_VEL
LIN {X 0,Y 508.121,Z 684.48,A -85,B 0,C 180,E1 -2932.977,E2 -2932.977} C_VEL
LIN {X 0,Y 499.836,Z 710.258,A -85,B 0,C 180,E1 -2934.047,E2 -2934.047} C_VEL
LIN {X 0,Y 497.751,Z 718.943,A -85,B 0,C 180,E1 -2934.415,E2 -2934.415} C_VEL
LIN {X 0,Y 496.996,Z 761.232,A -85,B 0,C 180,E1 -2935.076,E2 -2935.076} C_VEL
LIN {X 0,Y 496.1,Z 785.159,A -85,B 0,C 180,E1 -2935.664,E2 -2935.664} C_VEL
LIN {X 0,Y 495.065,Z 807.747,A -85,B 0,C 180,E1 -2936.435,E2 -2936.435} C_VEL
LIN {X 0,Y 493.81,Z 829.795,A -85,B 0,C 180,E1 -2937.412,E2 -2937.412} C_VEL
LIN {X 0,Y 492.4,Z 850.479,A -85,B 0,C 180,E1 -2938.542,E2 -2938.542} C_VEL
LIN {X 0,Y 491.075,Z 867.33,A -85,B 0,C 180,E1 -2939.687,E2 -2939.687} C_VEL
LIN {X 0,Y 489.302,Z 885.09,A -85,B 0,C 180,E1 -2941.167,E2 -2941.167} C_VEL
LIN {X 0,Y 487.436,Z 903.498,A -85,B 0,C 180,E1 -2942.976,E2 -2942.976} C_VEL
LIN {X 0,Y 485.711,Z 920.23,A -85,B 0,C 180,E1 -2944.908,E2 -2944.908} C_VEL
LIN {X 0,Y 484.158,Z 935.911,A -85,B 0,C 180,E1 -2947.026,E2 -2947.026} C_VEL
LIN {X 0,Y 482.865,Z 950.066,A -85,B 0,C 180,E1 -2949.262,E2 -2949.262} C_VEL
LIN {X 0,Y 481.83,Z 962.743,A -85,B 0,C 180,E1 -2951.613,E2 -2951.613} C_VEL
LIN {X 0,Y 480.999,Z 974.607,A -85,B 0,C 180,E1 -2954.246,E2 -2954.246} C_VEL
LIN {X 0,Y 480.458,Z 984.342,A -85,B 0,C 180,E1 -2956.889,E2 -2956.889} C_VEL
LIN {X 0,Y 480.144,Z 992.203,A -85,B 0,C 180,E1 -2959.562,E2 -2959.562} C_VEL
LIN {X 0,Y 479.975,Z 998.151,A -85,B 0,C 180,E1 -2962.218,E2 -2962.218} C_VEL
LIN {X 0,Y 479.909,Z 1002.133,A -85,B 0,C 180,E1 -2964.74,E2 -2964.74} C_VEL
LIN {X 0,Y 479.895,Z 1004.437,A -85,B 0,C 180,E1 -2967.133,E2 -2967.133} C_VEL
LIN {X 0,Y 479.893,Z 1005.391,A -85,B 0,C 180,E1 -2969.403,E2 -2969.403} C_VEL
LIN {X 0,Y 479.905,Z 1005.048,A -85,B 0,C 180,E1 -2971.91,E2 -2971.91} C_VEL
LIN {X 0,Y 479.918,Z 1002.997,A -85,B 0,C 180,E1 -2974.54,E2 -2974.54} C_VEL
LIN {X 0,Y 479.953,Z 999.437,A -85,B 0,C 180,E1 -2977.06,E2 -2977.06} C_VEL
LIN {X 0,Y 480.063,Z 994.3,A -85,B 0,C 180,E1 -2979.591,E2 -2979.591} C_VEL
LIN {X 0,Y 480.324,Z 987.071,A -85,B 0,C 180,E1 -2982.258,E2 -2982.258} C_VEL
LIN {X 0,Y 480.802,Z 977.803,A -85,B 0,C 180,E1 -2984.943,E2 -2984.943} C_VEL
LIN {X 0,Y 481.519,Z 966.878,A -85,B 0,C 180,E1 -2987.523,E2 -2987.523} C_VEL
LIN {X 0,Y 482.502,Z 954.314,A -85,B 0,C 180,E1 -2989.994,E2 -2989.994} C_VEL
LIN {X 0,Y 483.776,Z 940.096,A -85,B 0,C 180,E1 -2992.351,E2 -2992.351} C_VEL
LIN {X 0,Y 485.29,Z 924.513,A -85,B 0,C 180,E1 -2994.547,E2 -2994.547} C_VEL
LIN {X 0,Y 486.949,Z 908.076,A -85,B 0,C 180,E1 -2996.525,E2 -2996.525} C_VEL
LIN {X 0,Y 488.772,Z 890.513,A -85,B 0,C 180,E1 -2998.332,E2 -2998.332} C_VEL
LIN {X 0,Y 490.622,Z 871.933,A -85,B 0,C 180,E1 -2999.953,E2 -2999.953} C_VEL
LIN {X 0,Y 492.056,Z 855.569,A -85,B 0,C 180,E1 -3001.141,E2 -3001.141} C_VEL
LIN {X 0,Y 493.643,Z 834.589,A -85,B 0,C 180,E1 -3002.393,E2 -3002.393} C_VEL
LIN {X 0,Y 495.133,Z 812.739,A -85,B 0,C 180,E1 -3003.455,E2 -3003.455} C_VEL
LIN {X 0,Y 496.417,Z 789.93,A -85,B 0,C 180,E1 -3004.326,E2 -3004.326} C_VEL
LIN {X 0,Y 497.491,Z 767.008,A -85,B 0,C 180,E1 -3004.963,E2 -3004.963} C_VEL
LIN {X 0,Y 498.141,Z 741.239,A -85,B 0,C 180,E1 -3005.431,E2 -3005.431} C_VEL
LIN {X 0,Y 498.567,Z 719.435,A -85,B 0,C 180,E1 -3005.774,E2 -3005.774} C_VEL
LIN {X 0,Y 503.253,Z 702.846,A -85,B 0,C 180,E1 -3006.515,E2 -3006.515} C_VEL
LIN {X 0,Y 509.872,Z 683.135,A -85,B 0,C 180,E1 -3007.297,E2 -3007.297} C_VEL
LIN {X 0,Y 516.469,Z 667.941,A -85,B 0,C 180,E1 -3007.787,E2 -3007.787} C_VEL
LIN {X 0,Y 521.463,Z 654.56,A -85,B 0,C 180,E1 -3008.266,E2 -3008.266} C_VEL
LIN {X 0,Y 530.083,Z 636.613,A -85,B 0,C 180,E1 -3008.772,E2 -3008.772} C_VEL
LIN {X 0,Y 544.48,Z 611.009,A -85,B 0,C 180,E1 -3009.312,E2 -3009.312} C_VEL
LIN {X 0,Y 556.486,Z 589.897,A -85,B 0,C 180,E1 -3009.631,E2 -3009.631} C_VEL
LIN {X 0,Y 558.998,Z 585.027,A -85,B 0,C 180,E1 -3009.684,E2 -3009.684} C_VEL
LIN {X 0,Y 564.237,Z 571.353,A -85,B 0,C 180,E1 -3010.035,E2 -3010.035} C_VEL
LIN {X 0,Y 568.184,Z 561.557,A -85,B 0,C 180,E1 -3010.227,E2 -3010.227} C_VEL
LIN {X 0,Y 564.757,Z 561.53,A -85,B 0,C 180,E1 -3010.735,E2 -3010.735} C_VEL
LIN {X 0,Y 559.025,Z 560.212,A -85,B 0,C 180,E1 -3011.306,E2 -3011.306} C_VEL
LIN {X 0,Y 548.27,Z 556.129,A -85,B 0,C 180,E1 -3012.39,E2 -3012.39} C_VEL
LIN {X 0,Y 538.353,Z 550.39,A -85,B 0,C 180,E1 -3013.587,E2 -3013.587} C_VEL
LIN {X 0,Y 529.92,Z 543.337,A -85,B 0,C 180,E1 -3014.811,E2 -3014.811} C_VEL
LIN {X 0,Y 522.447,Z 534.272,A -85,B 0,C 180,E1 -3016.149,E2 -3016.149} C_VEL
LIN {X 0,Y 516.988,Z 524.522,A -85,B 0,C 180,E1 -3017.398,E2 -3017.398} C_VEL
LIN {X 0,Y 512.78,Z 513.028,A -85,B 0,C 180,E1 -3018.698,E2 -3018.698} C_VEL
LIN {X 0,Y 510.062,Z 499.55,A -85,B 0,C 180,E1 -3020.037,E2 -3020.037} C_VEL
LIN {X 0,Y 508.869,Z 483.471,A -85,B 0,C 180,E1 -3021.445,E2 -3021.445} C_VEL
LIN {X 0,Y 509.56,Z 463.804,A -85,B 0,C 180,E1 -3022.959,E2 -3022.959} C_VEL
LIN {X 0,Y 512.538,Z 427.742,A -85,B 0,C 180,E1 -3025.607,E2 -3025.607} C_VEL
LIN {X 0,Y 502.283,Z 409.024,A -85,B 0,C 180,E1 -3028.698,E2 -3028.698} C_VEL
LIN {X 0,Y 494.33,Z 394.948,A -85,B 0,C 180,E1 -3031.224,E2 -3031.224} C_VEL
LIN {X 0,Y 488.628,Z 385.13,A -85,B 0,C 180,E1 -3033.114,E2 -3033.114} C_VEL
LIN {X 0,Y 485.8,Z 380.212,A -85,B 0,C 180,E1 -3034.081,E2 -3034.081} C_VEL
LIN {X 0,Y 483.851,Z 376.481,A -85,B 0,C 180,E1 -3034.806,E2 -3034.806} C_VEL
LIN {X 0,Y 481.481,Z 373.009,A -85,B 0,C 180,E1 -3035.591,E2 -3035.591} C_VEL
LIN {X 0,Y 480.891,Z 370.83,A -85,B 0,C 180,E1 -3035.951,E2 -3035.951} C_VEL
LIN {X 0,Y 480.843,Z 370.836,A -85,B 0,C 180,E1 -3039.426,E2 -3039.426} C_VEL
LIN {X 0,Y 480.872,Z 370.833,A -85,B 0,C 180,E1 -3043.077,E2 -3043.077} C_VEL
LIN {X 0,Y 480.893,Z 370.832,A -85,B 0,C 180,E1 -3046.667,E2 -3046.667} C_VEL
LIN {X 0,Y 480.892,Z 370.833,A -85,B 0,C 180,E1 -3050.305,E2 -3050.305} C_VEL
LIN {X 0,Y 480.854,Z 370.836,A -85,B 0,C 180,E1 -3053.913,E2 -3053.913} C_VEL
LIN {X 0,Y 480.866,Z 370.839,A -85,B 0,C 180,E1 -3057.617,E2 -3057.617} C_VEL
LIN {X 0,Y 480.895,Z 370.835,A -85,B 0,C 180,E1 -3061.192,E2 -3061.192} C_VEL
LIN {X 0,Y 480.894,Z 370.834,A -85,B 0,C 180,E1 -3065.01,E2 -3065.01} C_VEL
LIN {X 0,Y 480.86,Z 370.839,A -85,B 0,C 180,E1 -3068.61,E2 -3068.61} C_VEL
LIN {X 0,Y 480.862,Z 370.839,A -85,B 0,C 180,E1 -3072.367,E2 -3072.367} C_VEL
LIN {X 0,Y 480.892,Z 370.832,A -85,B 0,C 180,E1 -3075.93,E2 -3075.93} C_VEL
LIN {X 0,Y 480.889,Z 370.834,A -85,B 0,C 180,E1 -3079.684,E2 -3079.684} C_VEL
LIN {X 0,Y 480.867,Z 370.834,A -85,B 0,C 180,E1 -3083.214,E2 -3083.214} C_VEL
LIN {X 0,Y 480.857,Z 370.834,A -85,B 0,C 180,E1 -3086.956,E2 -3086.956} C_VEL
LIN {X 0,Y 480.893,Z 370.832,A -85,B 0,C 180,E1 -3090.486,E2 -3090.486} C_VEL
LIN {X 0,Y 480.885,Z 370.83,A -85,B 0,C 180,E1 -3094.155,E2 -3094.155} C_VEL
LIN {X 0,Y 480.872,Z 370.819,A -85,B 0,C 180,E1 -3097.684,E2 -3097.684} C_VEL
LIN {X 0,Y 480.845,Z 370.827,A -85,B 0,C 180,E1 -3101.395,E2 -3101.395} C_VEL
LIN {X 0,Y 480.89,Z 370.838,A -85,B 0,C 180,E1 -3105.015,E2 -3105.015} C_VEL
LIN {X 0,Y 480.889,Z 370.834,A -85,B 0,C 180,E1 -3108.642,E2 -3108.642} C_VEL
LIN {X 0,Y 480.881,Z 370.828,A -85,B 0,C 180,E1 -3112.196,E2 -3112.196} C_VEL
LIN {X 0,Y 480.913,Z 371.049,A -85,B 0,C 180,E1 -3112.471,E2 -3112.471} C_VEL
LIN {X 0,Y 490.058,Z 394.023,A -85,B 0,C 180,E1 -3115.018,E2 -3115.018} C_VEL
LIN {X 0,Y 493.458,Z 403.6,A -85,B 0,C 180,E1 -3116.06,E2 -3116.06} C_VEL
LIN {X 0,Y 493.054,Z 413.215,A -85,B 0,C 180,E1 -3116.804,E2 -3116.804} C_VEL
LIN {X 0,Y 491.911,Z 419.851,A -85,B 0,C 180,E1 -3117.254,E2 -3117.254} C_VEL
LIN {X 0,Y 485.741,Z 438.301,A -85,B 0,C 180,E1 -3118.261,E2 -3118.261} C_VEL
LIN {X 0,Y 484.851,Z 444.041,A -85,B 0,C 180,E1 -3118.649,E2 -3118.649} C_VEL
LIN {X 0,Y 483.899,Z 479.277,A -85,B 0,C 180,E1 -3121.221,E2 -3121.221} C_VEL
LIN {X 0,Y 483.984,Z 484.681,A -85,B 0,C 180,E1 -3121.557,E2 -3121.557} C_VEL
LIN {X 0,Y 485.045,Z 492.92,A -85,B 0,C 180,E1 -3121.766,E2 -3121.766} C_VEL
LIN {X 0,Y 482.322,Z 692.399,A -85,B 0,C 180,E1 -3124.914,E2 -3124.914} C_VEL
LIN {X 0,Y 481.927,Z 710.874,A -85,B 0,C 180,E1 -3125.419,E2 -3125.419} C_VEL
LIN {X 0,Y 481.278,Z 728.911,A -85,B 0,C 180,E1 -3126.135,E2 -3126.135} C_VEL
LIN {X 0,Y 480.404,Z 745.922,A -85,B 0,C 180,E1 -3127.031,E2 -3127.031} C_VEL
LIN {X 0,Y 479.422,Z 761.667,A -85,B 0,C 180,E1 -3128.08,E2 -3128.08} C_VEL
LIN {X 0,Y 478.326,Z 777.432,A -85,B 0,C 180,E1 -3129.377,E2 -3129.377} C_VEL
LIN {X 0,Y 477.153,Z 792.165,A -85,B 0,C 180,E1 -3130.856,E2 -3130.856} C_VEL
LIN {X 0,Y 476.019,Z 805.815,A -85,B 0,C 180,E1 -3132.521,E2 -3132.521} C_VEL
LIN {X 0,Y 474.959,Z 818.261,A -85,B 0,C 180,E1 -3134.368,E2 -3134.368} C_VEL
LIN {X 0,Y 474.073,Z 829.124,A -85,B 0,C 180,E1 -3136.337,E2 -3136.337} C_VEL
LIN {X 0,Y 473.387,Z 838.454,A -85,B 0,C 180,E1 -3138.425,E2 -3138.425} C_VEL
LIN {X 0,Y 472.867,Z 846.245,A -85,B 0,C 180,E1 -3140.63,E2 -3140.63} C_VEL
LIN {X 0,Y 472.553,Z 852.443,A -85,B 0,C 180,E1 -3142.951,E2 -3142.951} C_VEL
LIN {X 0,Y 472.396,Z 856.768,A -85,B 0,C 180,E1 -3145.265,E2 -3145.265} C_VEL
LIN {X 0,Y 472.307,Z 859.362,A -85,B 0,C 180,E1 -3147.574,E2 -3147.574} C_VEL
LIN {X 0,Y 472.283,Z 860.301,A -85,B 0,C 180,E1 -3149.879,E2 -3149.879} C_VEL
LIN {X 0,Y 472.307,Z 859.542,A -85,B 0,C 180,E1 -3152.306,E2 -3152.306} C_VEL
LIN {X 0,Y 472.391,Z 857.102,A -85,B 0,C 180,E1 -3154.614,E2 -3154.614} C_VEL
LIN {X 0,Y 472.536,Z 852.929,A -85,B 0,C 180,E1 -3156.928,E2 -3156.928} C_VEL
LIN {X 0,Y 472.816,Z 847.273,A -85,B 0,C 180,E1 -3159.126,E2 -3159.126} C_VEL
LIN {X 0,Y 473.294,Z 839.767,A -85,B 0,C 180,E1 -3161.331,E2 -3161.331} C_VEL
LIN {X 0,Y 473.944,Z 830.749,A -85,B 0,C 180,E1 -3163.419,E2 -3163.419} C_VEL
LIN {X 0,Y 474.783,Z 820.235,A -85,B 0,C 180,E1 -3165.388,E2 -3165.388} C_VEL
LIN {X 0,Y 475.808,Z 808.2,A -85,B 0,C 180,E1 -3167.236,E2 -3167.236} C_VEL
LIN {X 0,Y 476.902,Z 795.077,A -85,B 0,C 180,E1 -3168.901,E2 -3168.901} C_VEL
LIN {X 0,Y 478.039,Z 780.985,A -85,B 0,C 180,E1 -3170.381,E2 -3170.381} C_VEL
LIN {X 0,Y 479.13,Z 766.031,A -85,B 0,C 180,E1 -3171.677,E2 -3171.677} C_VEL
LIN {X 0,Y 480.145,Z 750.31,A -85,B 0,C 180,E1 -3172.789,E2 -3172.789} C_VEL
LIN {X 0,Y 481.042,Z 733.889,A -85,B 0,C 180,E1 -3173.716,E2 -3173.716} C_VEL
LIN {X 0,Y 481.771,Z 715.966,A -85,B 0,C 180,E1 -3174.492,E2 -3174.492} C_VEL
LIN {X 0,Y 482.248,Z 697.603,A -85,B 0,C 180,E1 -3175.057,E2 -3175.057} C_VEL
LIN {X 0,Y 482.513,Z 675.621,A -85,B 0,C 180,E1 -3175.471,E2 -3175.471} C_VEL
LIN {X 0,Y 484.906,Z 490.248,A -85,B 0,C 180,E1 -3178.379,E2 -3178.379} C_VEL
LIN {X 0,Y 483.877,Z 483.685,A -85,B 0,C 180,E1 -3178.574,E2 -3178.574} C_VEL
LIN {X 0,Y 484.531,Z 452.773,A -85,B 0,C 180,E1 -3180.782,E2 -3180.782} C_VEL
LIN {X 0,Y 486.486,Z 406.561,A -85,B 0,C 180,E1 -3184.36,E2 -3184.36} C_VEL
LIN {X 0,Y 478.629,Z 385.753,A -85,B 0,C 180,E1 -3186.688,E2 -3186.688} C_VEL
LIN {X 0,Y 472.93,Z 372.068,A -85,B 0,C 180,E1 -3188.25,E2 -3188.25} C_VEL
LIN {X 0,Y 472.943,Z 371.815,A -85,B 0,C 180,E1 -3191.432,E2 -3191.432} C_VEL
LIN {X 0,Y 472.92,Z 371.81,A -85,B 0,C 180,E1 -3194.923,E2 -3194.923} C_VEL
LIN {X 0,Y 472.926,Z 372.029,A -85,B 0,C 180,E1 -3198.321,E2 -3198.321} C_VEL
LIN {X 0,Y 474.301,Z 375.435,A -85,B 0,C 180,E1 -3198.815,E2 -3198.815} C_VEL
LIN {X 0,Y 482.343,Z 394.347,A -85,B 0,C 180,E1 -3201.503,E2 -3201.503} C_VEL
LIN {X 0,Y 489.145,Z 411.675,A -85,B 0,C 180,E1 -3203.79,E2 -3203.79} C_VEL
LIN {X 0,Y 486.529,Z 453.634,A -85,B 0,C 180,E1 -3207.423,E2 -3207.423} C_VEL
LIN {X 0,Y 484.028,Z 496.952,A -85,B 0,C 180,E1 -3211.094,E2 -3211.094} C_VEL
LIN {X 0,Y 481.591,Z 543.039,A -85,B 0,C 180,E1 -3214.942,E2 -3214.942} C_VEL
LIN {X 0,Y 479.439,Z 588.913,A -85,B 0,C 180,E1 -3218.723,E2 -3218.723} C_VEL
LIN {X 0,Y 479.214,Z 596.451,A -85,B 0,C 180,E1 -3219.309,E2 -3219.309} C_VEL
LIN {X 0,Y 479.946,Z 604.036,A -85,B 0,C 180,E1 -3219.493,E2 -3219.493} C_VEL
LIN {X 0,Y 477.475,Z 741.389,A -85,B 0,C 180,E1 -3221.969,E2 -3221.969} C_VEL
LIN {X 0,Y 477.147,Z 758.335,A -85,B 0,C 180,E1 -3222.512,E2 -3222.512} C_VEL
LIN {X 0,Y 476.662,Z 773.943,A -85,B 0,C 180,E1 -3223.248,E2 -3223.248} C_VEL
LIN {X 0,Y 476.054,Z 789.262,A -85,B 0,C 180,E1 -3224.217,E2 -3224.217} C_VEL
LIN {X 0,Y 475.383,Z 803.167,A -85,B 0,C 180,E1 -3225.355,E2 -3225.355} C_VEL
LIN {X 0,Y 474.703,Z 816.476,A -85,B 0,C 180,E1 -3226.727,E2 -3226.727} C_VEL
LIN {X 0,Y 474.094,Z 827.809,A -85,B 0,C 180,E1 -3228.195,E2 -3228.195} C_VEL
LIN {X 0,Y 473.553,Z 838.389,A -85,B 0,C 180,E1 -3229.907,E2 -3229.907} C_VEL
LIN {X 0,Y 473.156,Z 846.647,A -85,B 0,C 180,E1 -3231.616,E2 -3231.616} C_VEL
LIN {X 0,Y 472.866,Z 853.899,A -85,B 0,C 180,E1 -3233.565,E2 -3233.565} C_VEL
LIN {X 0,Y 472.691,Z 859.031,A -85,B 0,C 180,E1 -3235.511,E2 -3235.511} C_VEL
LIN {X 0,Y 472.636,Z 862.383,A -85,B 0,C 180,E1 -3237.453,E2 -3237.453} C_VEL
LIN {X 0,Y 472.622,Z 864.006,A -85,B 0,C 180,E1 -3239.394,E2 -3239.394} C_VEL
LIN {X 0,Y 472.686,Z 863.926,A -85,B 0,C 180,E1 -3241.454,E2 -3241.454} C_VEL
LIN {X 0,Y 472.786,Z 862.074,A -85,B 0,C 180,E1 -3243.434,E2 -3243.434} C_VEL
LIN {X 0,Y 473.005,Z 858.347,A -85,B 0,C 180,E1 -3245.458,E2 -3245.458} C_VEL
LIN {X 0,Y 473.297,Z 853.225,A -85,B 0,C 180,E1 -3247.282,E2 -3247.282} C_VEL
LIN {X 0,Y 473.744,Z 846.26,A -85,B 0,C 180,E1 -3249.107,E2 -3249.107} C_VEL
LIN {X 0,Y 474.281,Z 837.789,A -85,B 0,C 180,E1 -3250.814,E2 -3250.814} C_VEL
LIN {X 0,Y 474.923,Z 827.815,A -85,B 0,C 180,E1 -3252.4,E2 -3252.4} C_VEL
LIN {X 0,Y 475.62,Z 817.047,A -85,B 0,C 180,E1 -3253.776,E2 -3253.776} C_VEL
LIN {X 0,Y 476.366,Z 804.133,A -85,B 0,C 180,E1 -3255.09,E2 -3255.09} C_VEL
LIN {X 0,Y 477.009,Z 791.415,A -85,B 0,C 180,E1 -3256.125,E2 -3256.125} C_VEL
LIN {X 0,Y 477.566,Z 776.83,A -85,B 0,C 180,E1 -3257.044,E2 -3257.044} C_VEL
LIN {X 0,Y 477.999,Z 761.408,A -85,B 0,C 180,E1 -3257.77,E2 -3257.77} C_VEL
LIN {X 0,Y 478.207,Z 744.843,A -85,B 0,C 180,E1 -3258.289,E2 -3258.289} C_VEL
LIN {X 0,Y 480.383,Z 680.152,A -85,B 0,C 180,E1 -3259.768,E2 -3259.768} C_VEL
LIN {X 0,Y 484.049,Z 612.56,A -85,B 0,C 180,E1 -3261.413,E2 -3261.413} C_VEL
LIN {X 0,Y 486.077,Z 605.975,A -85,B 0,C 180,E1 -3261.858,E2 -3261.858} C_VEL
LIN {X 0,Y 490.908,Z 565.427,A -85,B 0,C 180,E1 -3265.646,E2 -3265.646} C_VEL
LIN {X 0,Y 496.917,Z 528.804,A -85,B 0,C 180,E1 -3269.271,E2 -3269.271} C_VEL
LIN {X 0,Y 502.767,Z 503.589,A -85,B 0,C 180,E1 -3271.937,E2 -3271.937} C_VEL
LIN {X 0,Y 508.777,Z 484.825,A -85,B 0,C 180,E1 -3274.061,E2 -3274.061} C_VEL
LIN {X 0,Y 515.474,Z 469.876,A -85,B 0,C 180,E1 -3275.886,E2 -3275.886} C_VEL
LIN {X 0,Y 508.579,Z 481.042,A -85,B 0,C 180,E1 -3277.228,E2 -3277.228} C_VEL
LIN {X 0,Y 504.479,Z 491.152,A -85,B 0,C 180,E1 -3278.486,E2 -3278.486} C_VEL
LIN {X 0,Y 502.432,Z 501.84,A -85,B 0,C 180,E1 -3279.85,E2 -3279.85} C_VEL
LIN {X 0,Y 502.673,Z 512.146,A -85,B 0,C 180,E1 -3281.176,E2 -3281.176} C_VEL
LIN {X 0,Y 505.16,Z 522.491,A -85,B 0,C 180,E1 -3282.526,E2 -3282.526} C_VEL
LIN {X 0,Y 509.764,Z 532.283,A -85,B 0,C 180,E1 -3283.818,E2 -3283.818} C_VEL
LIN {X 0,Y 516.639,Z 541.742,A -85,B 0,C 180,E1 -3285.098,E2 -3285.098} C_VEL
LIN {X 0,Y 524.862,Z 549.851,A -85,B 0,C 180,E1 -3286.219,E2 -3286.219} C_VEL
LIN {X 0,Y 535.655,Z 557.683,A -85,B 0,C 180,E1 -3287.344,E2 -3287.344} C_VEL
LIN {X 0,Y 548.32,Z 564.319,A -85,B 0,C 180,E1 -3288.385,E2 -3288.385} C_VEL
LIN {X 0,Y 558.973,Z 568.167,A -85,B 0,C 180,E1 -3289.168,E2 -3289.168} C_VEL
LIN {X 0,Y 560.111,Z 568.68,A -85,B 0,C 180,E1 -3289.29,E2 -3289.29} C_VEL
LIN {X 0,Y 553.967,Z 582.808,A -85,B 0,C 180,E1 -3289.679,E2 -3289.679} C_VEL
LIN {X 0,Y 551.879,Z 586.702,A -85,B 0,C 180,E1 -3289.768,E2 -3289.768} C_VEL
LIN {X 0,Y 527.647,Z 625.749,A -85,B 0,C 180,E1 -3290.664,E2 -3290.664} C_VEL
LIN {X 0,Y 517.206,Z 645.161,A -85,B 0,C 180,E1 -3291.218,E2 -3291.218} C_VEL
LIN {X 0,Y 510.459,Z 660.79,A -85,B 0,C 180,E1 -3291.759,E2 -3291.759} C_VEL
LIN {X 0,Y 507.462,Z 668.825,A -85,B 0,C 180,E1 -3292.067,E2 -3292.067} C_VEL
LIN {X 0,Y 500.634,Z 684.358,A -85,B 0,C 180,E1 -3292.616,E2 -3292.616} C_VEL
LIN {X 0,Y 492.38,Z 710.255,A -85,B 0,C 180,E1 -3293.705,E2 -3293.705} C_VEL
LIN {X 0,Y 490.627,Z 717.519,A -85,B 0,C 180,E1 -3294.008,E2 -3294.008} C_VEL
LIN {X 0,Y 489.913,Z 751.738,A -85,B 0,C 180,E1 -3294.526,E2 -3294.526} C_VEL
LIN {X 0,Y 489.086,Z 775.768,A -85,B 0,C 180,E1 -3295.044,E2 -3295.044} C_VEL
LIN {X 0,Y 488.058,Z 798.25,A -85,B 0,C 180,E1 -3295.749,E2 -3295.749} C_VEL
LIN {X 0,Y 486.775,Z 820.633,A -85,B 0,C 180,E1 -3296.67,E2 -3296.67} C_VEL
LIN {X 0,Y 485.37,Z 841.759,A -85,B 0,C 180,E1 -3297.755,E2 -3297.755} C_VEL
LIN {X 0,Y 483.822,Z 862.563,A -85,B 0,C 180,E1 -3299.051,E2 -3299.051} C_VEL
LIN {X 0,Y 482.239,Z 882.062,A -85,B 0,C 180,E1 -3300.499,E2 -3300.499} C_VEL
LIN {X 0,Y 480.818,Z 896.962,A -85,B 0,C 180,E1 -3301.848,E2 -3301.848} C_VEL
LIN {X 0,Y 478.998,Z 913.535,A -85,B 0,C 180,E1 -3303.668,E2 -3303.668} C_VEL
LIN {X 0,Y 477.219,Z 929.77,A -85,B 0,C 180,E1 -3305.754,E2 -3305.754} C_VEL
LIN {X 0,Y 475.664,Z 944.85,A -85,B 0,C 180,E1 -3308.027,E2 -3308.027} C_VEL
LIN {X 0,Y 474.397,Z 958.32,A -85,B 0,C 180,E1 -3310.42,E2 -3310.42} C_VEL
LIN {X 0,Y 473.375,Z 970.765,A -85,B 0,C 180,E1 -3313.053,E2 -3313.053} C_VEL
LIN {X 0,Y 472.692,Z 980.991,A -85,B 0,C 180,E1 -3315.671,E2 -3315.671} C_VEL
LIN {X 0,Y 472.276,Z 989.215,A -85,B 0,C 180,E1 -3318.273,E2 -3318.273} C_VEL
LIN {X 0,Y 472.054,Z 995.663,A -85,B 0,C 180,E1 -3320.859,E2 -3320.859} C_VEL
LIN {X 0,Y 471.953,Z 1000.566,A -85,B 0,C 180,E1 -3323.512,E2 -3323.512} C_VEL
LIN {X 0,Y 471.912,Z 1003.833,A -85,B 0,C 180,E1 -3326.234,E2 -3326.234} C_VEL
LIN {X 0,Y 471.908,Z 1005.251,A -85,B 0,C 180,E1 -3328.786,E2 -3328.786} C_VEL
LIN {X 0,Y 471.908,Z 1005.316,A -85,B 0,C 180,E1 -3331.214,E2 -3331.214} C_VEL
LIN {X 0,Y 471.912,Z 1003.721,A -85,B 0,C 180,E1 -3333.887,E2 -3333.887} C_VEL
LIN {X 0,Y 471.958,Z 1000.262,A -85,B 0,C 180,E1 -3336.691,E2 -3336.691} C_VEL
LIN {X 0,Y 472.065,Z 995.131,A -85,B 0,C 180,E1 -3339.386,E2 -3339.386} C_VEL
LIN {X 0,Y 472.303,Z 988.506,A -85,B 0,C 180,E1 -3341.973,E2 -3341.973} C_VEL
LIN {X 0,Y 472.718,Z 980.544,A -85,B 0,C 180,E1 -3344.453,E2 -3344.453} C_VEL
LIN {X 0,Y 473.419,Z 970.236,A -85,B 0,C 180,E1 -3347.071,E2 -3347.071} C_VEL
LIN {X 0,Y 474.457,Z 957.675,A -85,B 0,C 180,E1 -3349.705,E2 -3349.705} C_VEL
LIN {X 0,Y 475.741,Z 944.081,A -85,B 0,C 180,E1 -3352.098,E2 -3352.098} C_VEL
LIN {X 0,Y 477.317,Z 928.88,A -85,B 0,C 180,E1 -3354.372,E2 -3354.372} C_VEL
LIN {X 0,Y 479.256,Z 911.214,A -85,B 0,C 180,E1 -3356.608,E2 -3356.608} C_VEL
LIN {X 0,Y 481.037,Z 894.883,A -85,B 0,C 180,E1 -3358.356,E2 -3358.356} C_VEL
LIN {X 0,Y 482.736,Z 876.776,A -85,B 0,C 180,E1 -3359.945,E2 -3359.945} C_VEL
LIN {X 0,Y 484.579,Z 856.207,A -85,B 0,C 180,E1 -3361.468,E2 -3361.468} C_VEL
LIN {X 0,Y 486.307,Z 835.108,A -85,B 0,C 180,E1 -3362.764,E2 -3362.764} C_VEL
LIN {X 0,Y 487.946,Z 812.834,A -85,B 0,C 180,E1 -3363.873,E2 -3363.873} C_VEL
LIN {X 0,Y 489.351,Z 789.843,A -85,B 0,C 180,E1 -3364.77,E2 -3364.77} C_VEL
LIN {X 0,Y 490.496,Z 767.422,A -85,B 0,C 180,E1 -3365.41,E2 -3365.41} C_VEL
LIN {X 0,Y 491.23,Z 742.766,A -85,B 0,C 180,E1 -3365.881,E2 -3365.881} C_VEL
LIN {X 0,Y 491.813,Z 718.571,A -85,B 0,C 180,E1 -3366.271,E2 -3366.271} C_VEL
LIN {X 0,Y 496.582,Z 702.135,A -85,B 0,C 180,E1 -3367.015,E2 -3367.015} C_VEL
LIN {X 0,Y 503.252,Z 682.422,A -85,B 0,C 180,E1 -3367.801,E2 -3367.801} C_VEL
LIN {X 0,Y 509.895,Z 667.23,A -85,B 0,C 180,E1 -3368.29,E2 -3368.29} C_VEL
LIN {X 0,Y 515.345,Z 652.827,A -85,B 0,C 180,E1 -3368.805,E2 -3368.805} C_VEL
LIN {X 0,Y 523.984,Z 635.03,A -85,B 0,C 180,E1 -3369.31,E2 -3369.31} C_VEL
LIN {X 0,Y 537.678,Z 610.722,A -85,B 0,C 180,E1 -3369.825,E2 -3369.825} C_VEL
LIN {X 0,Y 553.576,Z 583.876,A -85,B 0,C 180,E1 -3370.286,E2 -3370.286} C_VEL
LIN {X 0,Y 559.993,Z 568.931,A -85,B 0,C 180,E1 -3370.705,E2 -3370.705} C_VEL
LIN {X 0,Y 560.085,Z 568.428,A -85,B 0,C 180,E1 -3370.729,E2 -3370.729} C_VEL
LIN {X 0,Y 547.965,Z 564.605,A -85,B 0,C 180,E1 -3371.887,E2 -3371.887} C_VEL
LIN {X 0,Y 537.001,Z 559.071,A -85,B 0,C 180,E1 -3373.124,E2 -3373.124} C_VEL
LIN {X 0,Y 527.658,Z 552.152,A -85,B 0,C 180,E1 -3374.408,E2 -3374.408} C_VEL
LIN {X 0,Y 519.827,Z 543.862,A -85,B 0,C 180,E1 -3375.717,E2 -3375.717} C_VEL
LIN {X 0,Y 513.481,Z 534.277,A -85,B 0,C 180,E1 -3377.038,E2 -3377.038} C_VEL
LIN {X 0,Y 508.431,Z 522.875,A -85,B 0,C 180,E1 -3378.417,E2 -3378.417} C_VEL
LIN {X 0,Y 504.993,Z 509.885,A -85,B 0,C 180,E1 -3379.8,E2 -3379.8} C_VEL
LIN {X 0,Y 503.073,Z 494.448,A -85,B 0,C 180,E1 -3381.24,E2 -3381.24} C_VEL
LIN {X 0,Y 502.892,Z 478.099,A -85,B 0,C 180,E1 -3382.599,E2 -3382.599} C_VEL
LIN {X 0,Y 506.613,Z 432.281,A -85,B 0,C 180,E1 -3386.009,E2 -3386.009} C_VEL
LIN {X 0,Y 496.473,Z 413.761,A -85,B 0,C 180,E1 -3389.1,E2 -3389.1} C_VEL
LIN {X 0,Y 488.881,Z 400.321,A -85,B 0,C 180,E1 -3391.541,E2 -3391.541} C_VEL
LIN {X 0,Y 483.544,Z 391.029,A -85,B 0,C 180,E1 -3393.34,E2 -3393.34} C_VEL
LIN {X 0,Y 480.609,Z 385.947,A -85,B 0,C 180,E1 -3394.36,E2 -3394.36} C_VEL
LIN {X 0,Y 478.078,Z 381.48,A -85,B 0,C 180,E1 -3395.274,E2 -3395.274} C_VEL
LIN {X 0,Y 476.061,Z 377.894,A -85,B 0,C 180,E1 -3396.01,E2 -3396.01} C_VEL
LIN {X 0,Y 475.249,Z 376.503,A -85,B 0,C 180,E1 -3396.307,E2 -3396.307} C_VEL
LIN {X 0,Y 473.331,Z 373.445,A -85,B 0,C 180,E1 -3396.997,E2 -3396.997} C_VEL
LIN {X 0,Y 472.943,Z 371.819,A -85,B 0,C 180,E1 -3397.289,E2 -3397.289} C_VEL
LIN {X 0,Y 472.909,Z 371.823,A -85,B 0,C 180,E1 -3400.922,E2 -3400.922} C_VEL
LIN {X 0,Y 472.954,Z 371.817,A -85,B 0,C 180,E1 -3404.426,E2 -3404.426} C_VEL
LIN {X 0,Y 472.915,Z 371.825,A -85,B 0,C 180,E1 -3408.042,E2 -3408.042} C_VEL
LIN {X 0,Y 472.95,Z 371.823,A -85,B 0,C 180,E1 -3411.646,E2 -3411.646} C_VEL
LIN {X 0,Y 472.931,Z 371.829,A -85,B 0,C 180,E1 -3415.149,E2 -3415.149} C_VEL
LIN {X 0,Y 472.955,Z 371.824,A -85,B 0,C 180,E1 -3418.789,E2 -3418.789} C_VEL
LIN {X 0,Y 472.904,Z 371.831,A -85,B 0,C 180,E1 -3422.303,E2 -3422.303} C_VEL
LIN {X 0,Y 472.938,Z 371.825,A -85,B 0,C 180,E1 -3425.946,E2 -3425.946} C_VEL
LIN {X 0,Y 472.949,Z 371.826,A -85,B 0,C 180,E1 -3429.492,E2 -3429.492} C_VEL
LIN {X 0,Y 472.955,Z 371.823,A -85,B 0,C 180,E1 -3433.198,E2 -3433.198} C_VEL
LIN {X 0,Y 472.911,Z 371.827,A -85,B 0,C 180,E1 -3436.713,E2 -3436.713} C_VEL
LIN {X 0,Y 472.931,Z 371.825,A -85,B 0,C 180,E1 -3440.417,E2 -3440.417} C_VEL
LIN {X 0,Y 472.954,Z 371.82,A -85,B 0,C 180,E1 -3444.038,E2 -3444.038} C_VEL
LIN {X 0,Y 472.958,Z 371.817,A -85,B 0,C 180,E1 -3447.853,E2 -3447.853} C_VEL
LIN {X 0,Y 472.92,Z 371.818,A -85,B 0,C 180,E1 -3451.339,E2 -3451.339} C_VEL
LIN {X 0,Y 472.925,Z 371.811,A -85,B 0,C 180,E1 -3455.104,E2 -3455.104} C_VEL
LIN {X 0,Y 472.954,Z 371.818,A -85,B 0,C 180,E1 -3458.739,E2 -3458.739} C_VEL
LIN {X 0,Y 472.946,Z 371.801,A -85,B 0,C 180,E1 -3462.454,E2 -3462.454} C_VEL
LIN {X 0,Y 472.927,Z 371.822,A -85,B 0,C 180,E1 -3465.958,E2 -3465.958} C_VEL
LIN {X 0,Y 472.922,Z 371.83,A -85,B 0,C 180,E1 -3469.688,E2 -3469.688} C_VEL
LIN {X 0,Y 472.979,Z 372.026,A -85,B 0,C 180,E1 -3471.85,E2 -3471.85} C_VEL
LIN {X 0,Y 482.053,Z 394.518,A -85,B 0,C 180,E1 -3474.398,E2 -3474.398} C_VEL
LIN {X 0,Y 486.476,Z 406.449,A -85,B 0,C 180,E1 -3475.726,E2 -3475.726} C_VEL
LIN {X 0,Y 484.851,Z 444.041,A -85,B 0,C 180,E1 -3478.649,E2 -3478.649} C_VEL
LIN {X 0,Y 483.741,Z 450.772,A -85,B 0,C 180,E1 -3479.088,E2 -3479.088} C_VEL
LIN {X 0,Y 477.793,Z 469.537,A -85,B 0,C 180,E1 -3480.046,E2 -3480.046} C_VEL
LIN {X 0,Y 477.014,Z 475.411,A -85,B 0,C 180,E1 -3480.414,E2 -3480.414} C_VEL
LIN {X 0,Y 476.984,Z 485.748,A -85,B 0,C 180,E1 -3481.099,E2 -3481.099} C_VEL
LIN {X 0,Y 478.055,Z 493.944,A -85,B 0,C 180,E1 -3481.313,E2 -3481.313} C_VEL
LIN {X 0,Y 475.144,Z 693.538,A -85,B 0,C 180,E1 -3484.508,E2 -3484.508} C_VEL
LIN {X 0,Y 474.732,Z 712.079,A -85,B 0,C 180,E1 -3485.021,E2 -3485.021} C_VEL
LIN {X 0,Y 474.083,Z 729.438,A -85,B 0,C 180,E1 -3485.716,E2 -3485.716} C_VEL
LIN {X 0,Y 473.136,Z 747.158,A -85,B 0,C 180,E1 -3486.657,E2 -3486.657} C_VEL
LIN {X 0,Y 472.07,Z 763.383,A -85,B 0,C 180,E1 -3487.757,E2 -3487.757} C_VEL
LIN {X 0,Y 470.885,Z 779.379,A -85,B 0,C 180,E1 -3489.101,E2 -3489.101} C_VEL
LIN {X 0,Y 469.642,Z 793.99,A -85,B 0,C 180,E1 -3490.603,E2 -3490.603} C_VEL
LIN {X 0,Y 468.473,Z 807.072,A -85,B 0,C 180,E1 -3492.23,E2 -3492.23} C_VEL
LIN {X 0,Y 467.335,Z 819.52,A -85,B 0,C 180,E1 -3494.107,E2 -3494.107} C_VEL
LIN {X 0,Y 466.376,Z 830.386,A -85,B 0,C 180,E1 -3496.107,E2 -3496.107} C_VEL
LIN {X 0,Y 465.625,Z 839.717,A -85,B 0,C 180,E1 -3498.229,E2 -3498.229} C_VEL
LIN {X 0,Y 465.053,Z 847.51,A -85,B 0,C 180,E1 -3500.471,E2 -3500.471} C_VEL
LIN {X 0,Y 464.698,Z 853.708,A -85,B 0,C 180,E1 -3502.831,E2 -3502.831} C_VEL
LIN {X 0,Y 464.514,Z 858.032,A -85,B 0,C 180,E1 -3505.185,E2 -3505.185} C_VEL
LIN {X 0,Y 464.412,Z 860.626,A -85,B 0,C 180,E1 -3507.532,E2 -3507.532} C_VEL
LIN {X 0,Y 464.384,Z 861.564,A -85,B 0,C 180,E1 -3509.877,E2 -3509.877} C_VEL
LIN {X 0,Y 464.411,Z 860.805,A -85,B 0,C 180,E1 -3512.345,E2 -3512.345} C_VEL
LIN {X 0,Y 464.509,Z 858.329,A -85,B 0,C 180,E1 -3514.715,E2 -3514.715} C_VEL
LIN {X 0,Y 464.678,Z 854.191,A -85,B 0,C 180,E1 -3517.045,E2 -3517.045} C_VEL
LIN {X 0,Y 464.993,Z 848.534,A -85,B 0,C 180,E1 -3519.281,E2 -3519.281} C_VEL
LIN {X 0,Y 465.524,Z 841.026,A -85,B 0,C 180,E1 -3521.523,E2 -3521.523} C_VEL
LIN {X 0,Y 466.235,Z 832.004,A -85,B 0,C 180,E1 -3523.645,E2 -3523.645} C_VEL
LIN {X 0,Y 467.147,Z 821.486,A -85,B 0,C 180,E1 -3525.646,E2 -3525.646} C_VEL
LIN {X 0,Y 468.249,Z 809.448,A -85,B 0,C 180,E1 -3527.523,E2 -3527.523} C_VEL
LIN {X 0,Y 469.421,Z 796.321,A -85,B 0,C 180,E1 -3529.213,E2 -3529.213} C_VEL
LIN {X 0,Y 470.634,Z 782.223,A -85,B 0,C 180,E1 -3530.716,E2 -3530.716} C_VEL
LIN {X 0,Y 471.792,Z 767.262,A -85,B 0,C 180,E1 -3532.032,E2 -3532.032} C_VEL
LIN {X 0,Y 472.866,Z 751.532,A -85,B 0,C 180,E1 -3533.16,E2 -3533.16} C_VEL
LIN {X 0,Y 473.81,Z 735.098,A -85,B 0,C 180,E1 -3534.101,E2 -3534.101} C_VEL
LIN {X 0,Y 474.575,Z 717.152,A -85,B 0,C 180,E1 -3534.888,E2 -3534.888} C_VEL
LIN {X 0,Y 475.067,Z 698.808,A -85,B 0,C 180,E1 -3535.46,E2 -3535.46} C_VEL
LIN {X 0,Y 475.337,Z 676.816,A -85,B 0,C 180,E1 -3535.881,E2 -3535.881} C_VEL
LIN {X 0,Y 477.928,Z 491.505,A -85,B 0,C 180,E1 -3538.829,E2 -3538.829} C_VEL
LIN {X 0,Y 476.896,Z 484.705,A -85,B 0,C 180,E1 -3539.039,E2 -3539.039} C_VEL
LIN {X 0,Y 477.596,Z 453.5,A -85,B 0,C 180,E1 -3541.279,E2 -3541.279} C_VEL
LIN {X 0,Y 479.523,Z 409.513,A -85,B 0,C 180,E1 -3544.697,E2 -3544.697} C_VEL
LIN {X 0,Y 471.79,Z 389.311,A -85,B 0,C 180,E1 -3547.005,E2 -3547.005} C_VEL
LIN {X 0,Y 465.04,Z 373.096,A -85,B 0,C 180,E1 -3548.893,E2 -3548.893} C_VEL
LIN {X 0,Y 465.018,Z 372.814,A -85,B 0,C 180,E1 -3549.085,E2 -3549.085} C_VEL
LIN {X 0,Y 464.969,Z 372.818,A -85,B 0,C 180,E1 -3552.639,E2 -3552.639} C_VEL
LIN {X 0,Y 464.958,Z 372.82,A -85,B 0,C 180,E1 -3556.265,E2 -3556.265} C_VEL
LIN {X 0,Y 465.03,Z 372.971,A -85,B 0,C 180,E1 -3557.535,E2 -3557.535} C_VEL
LIN {X 0,Y 466.438,Z 376.52,A -85,B 0,C 180,E1 -3558.059,E2 -3558.059} C_VEL
LIN {X 0,Y 474.579,Z 395.456,A -85,B 0,C 180,E1 -3560.834,E2 -3560.834} C_VEL
LIN {X 0,Y 482.07,Z 414.361,A -85,B 0,C 180,E1 -3563.387,E2 -3563.387} C_VEL
LIN {X 0,Y 482.037,Z 418.68,A -85,B 0,C 180,E1 -3563.793,E2 -3563.793} C_VEL
LIN {X 0,Y 479.281,Z 460.626,A -85,B 0,C 180,E1 -3567.439,E2 -3567.439} C_VEL
LIN {X 0,Y 476.626,Z 504.012,A -85,B 0,C 180,E1 -3571.151,E2 -3571.151} C_VEL
LIN {X 0,Y 474.185,Z 547.99,A -85,B 0,C 180,E1 -3574.857,E2 -3574.857} C_VEL
LIN {X 0,Y 471.953,Z 593.357,A -85,B 0,C 180,E1 -3578.63,E2 -3578.63} C_VEL
LIN {X 0,Y 471.894,Z 597.312,A -85,B 0,C 180,E1 -3578.92,E2 -3578.92} C_VEL
LIN {X 0,Y 472.632,Z 604.93,A -85,B 0,C 180,E1 -3579.112,E2 -3579.112} C_VEL
LIN {X 0,Y 469.911,Z 742.542,A -85,B 0,C 180,E1 -3581.672,E2 -3581.672} C_VEL
LIN {X 0,Y 469.559,Z 759.656,A -85,B 0,C 180,E1 -3582.236,E2 -3582.236} C_VEL
LIN {X 0,Y 469.051,Z 775.059,A -85,B 0,C 180,E1 -3582.978,E2 -3582.978} C_VEL
LIN {X 0,Y 468.414,Z 790.206,A -85,B 0,C 180,E1 -3583.953,E2 -3583.953} C_VEL
LIN {X 0,Y 467.728,Z 803.747,A -85,B 0,C 180,E1 -3585.071,E2 -3585.071} C_VEL
LIN {X 0,Y 467.026,Z 816.624,A -85,B 0,C 180,E1 -3586.404,E2 -3586.404} C_VEL
LIN {X 0,Y 466.38,Z 828.04,A -85,B 0,C 180,E1 -3587.871,E2 -3587.871} C_VEL
LIN {X 0,Y 465.782,Z 838.803,A -85,B 0,C 180,E1 -3589.611,E2 -3589.611} C_VEL
LIN {X 0,Y 465.348,Z 847.296,A -85,B 0,C 180,E1 -3591.349,E2 -3591.349} C_VEL
LIN {X 0,Y 465.019,Z 854.701,A -85,B 0,C 180,E1 -3593.332,E2 -3593.332} C_VEL
LIN {X 0,Y 464.831,Z 859.77,A -85,B 0,C 180,E1 -3595.187,E2 -3595.187} C_VEL
LIN {X 0,Y 464.751,Z 863.518,A -85,B 0,C 180,E1 -3597.287,E2 -3597.287} C_VEL
LIN {X 0,Y 464.739,Z 865.319,A -85,B 0,C 180,E1 -3599.26,E2 -3599.26} C_VEL
LIN {X 0,Y 464.804,Z 865.366,A -85,B 0,C 180,E1 -3601.356,E2 -3601.356} C_VEL
LIN {X 0,Y 464.919,Z 863.737,A -85,B 0,C 180,E1 -3603.328,E2 -3603.328} C_VEL
LIN {X 0,Y 465.154,Z 860.079,A -85,B 0,C 180,E1 -3605.427,E2 -3605.427} C_VEL
LIN {X 0,Y 465.481,Z 855.142,A -85,B 0,C 180,E1 -3607.28,E2 -3607.28} C_VEL
LIN {X 0,Y 465.998,Z 847.821,A -85,B 0,C 180,E1 -3609.26,E2 -3609.26} C_VEL
LIN {X 0,Y 466.544,Z 840.098,A -85,B 0,C 180,E1 -3610.87,E2 -3610.87} C_VEL
LIN {X 0,Y 467.284,Z 829.484,A -85,B 0,C 180,E1 -3612.606,E2 -3612.606} C_VEL
LIN {X 0,Y 468.045,Z 818.525,A -85,B 0,C 180,E1 -3614.032,E2 -3614.032} C_VEL
LIN {X 0,Y 468.875,Z 805.387,A -85,B 0,C 180,E1 -3615.396,E2 -3615.396} C_VEL
LIN {X 0,Y 469.561,Z 792.543,A -85,B 0,C 180,E1 -3616.451,E2 -3616.451} C_VEL
LIN {X 0,Y 470.161,Z 777.939,A -85,B 0,C 180,E1 -3617.385,E2 -3617.385} C_VEL
LIN {X 0,Y 470.605,Z 762.542,A -85,B 0,C 180,E1 -3618.115,E2 -3618.115} C_VEL
LIN {X 0,Y 470.843,Z 746.052,A -85,B 0,C 180,E1 -3618.646,E2 -3618.646} C_VEL
LIN {X 0,Y 472.839,Z 691.917,A -85,B 0,C 180,E1 -3619.952,E2 -3619.952} C_VEL
LIN {X 0,Y 477.479,Z 614.972,A -85,B 0,C 180,E1 -3621.926,E2 -3621.926} C_VEL
LIN {X 0,Y 479.787,Z 607.741,A -85,B 0,C 180,E1 -3622.418,E2 -3622.418} C_VEL
LIN {X 0,Y 485.27,Z 566.431,A -85,B 0,C 180,E1 -3626.36,E2 -3626.36} C_VEL
LIN {X 0,Y 491.533,Z 532.306,A -85,B 0,C 180,E1 -3629.825,E2 -3629.825} C_VEL
LIN {X 0,Y 497.604,Z 508.783,A -85,B 0,C 180,E1 -3632.377,E2 -3632.377} C_VEL
LIN {X 0,Y 504.273,Z 490.13,A -85,B 0,C 180,E1 -3634.546,E2 -3634.546} C_VEL
LIN {X 0,Y 509.204,Z 479.821,A -85,B 0,C 180,E1 -3635.853,E2 -3635.853} C_VEL
LIN {X 0,Y 502.748,Z 490.417,A -85,B 0,C 180,E1 -3637.199,E2 -3637.199} C_VEL
LIN {X 0,Y 498.903,Z 500.256,A -85,B 0,C 180,E1 -3638.509,E2 -3638.509} C_VEL
LIN {X 0,Y 497.172,Z 510.556,A -85,B 0,C 180,E1 -3639.906,E2 -3639.906} C_VEL
LIN {X 0,Y 497.788,Z 520.773,A -85,B 0,C 180,E1 -3641.303,E2 -3641.303} C_VEL
LIN {X 0,Y 500.761,Z 530.956,A -85,B 0,C 180,E1 -3642.711,E2 -3642.711} C_VEL
LIN {X 0,Y 505.988,Z 540.761,A -85,B 0,C 180,E1 -3644.072,E2 -3644.072} C_VEL
LIN {X 0,Y 513.108,Z 549.717,A -85,B 0,C 180,E1 -3645.336,E2 -3645.336} C_VEL
LIN {X 0,Y 522.19,Z 557.984,A -85,B 0,C 180,E1 -3646.526,E2 -3646.526} C_VEL
LIN {X 0,Y 533.177,Z 565.428,A -85,B 0,C 180,E1 -3647.634,E2 -3647.634} C_VEL
LIN {X 0,Y 545.973,Z 571.783,A -85,B 0,C 180,E1 -3648.663,E2 -3648.663} C_VEL
LIN {X 0,Y 550.584,Z 573.703,A -85,B 0,C 180,E1 -3649.002,E2 -3649.002} C_VEL
LIN {X 0,Y 546.463,Z 582.923,A -85,B 0,C 180,E1 -3649.286,E2 -3649.286} C_VEL
LIN {X 0,Y 521.638,Z 622.666,A -85,B 0,C 180,E1 -3650.193,E2 -3650.193} C_VEL
LIN {X 0,Y 510.642,Z 642.995,A -85,B 0,C 180,E1 -3650.769,E2 -3650.769} C_VEL
LIN {X 0,Y 503.817,Z 658.61,A -85,B 0,C 180,E1 -3651.307,E2 -3651.307} C_VEL
LIN {X 0,Y 500.828,Z 666.711,A -85,B 0,C 180,E1 -3651.619,E2 -3651.619} C_VEL
LIN {X 0,Y 493.927,Z 682.277,A -85,B 0,C 180,E1 -3652.166,E2 -3652.166} C_VEL
LIN {X 0,Y 485.217,Z 709.173,A -85,B 0,C 180,E1 -3653.302,E2 -3653.302} C_VEL
LIN {X 0,Y 483.551,Z 716,A -85,B 0,C 180,E1 -3653.586,E2 -3653.586} C_VEL
LIN {X 0,Y 482.966,Z 729.546,A -85,B 0,C 180,E1 -3653.779,E2 -3653.779} C_VEL
LIN {X 0,Y 482.304,Z 761.787,A -85,B 0,C 180,E1 -3654.337,E2 -3654.337} C_VEL
LIN {X 0,Y 481.278,Z 785.096,A -85,B 0,C 180,E1 -3654.951,E2 -3654.951} C_VEL
LIN {X 0,Y 480.026,Z 807.897,A -85,B 0,C 180,E1 -3655.783,E2 -3655.783} C_VEL
LIN {X 0,Y 478.613,Z 830.013,A -85,B 0,C 180,E1 -3656.815,E2 -3656.815} C_VEL
LIN {X 0,Y 477.072,Z 850.347,A -85,B 0,C 180,E1 -3657.978,E2 -3657.978} C_VEL
LIN {X 0,Y 475.482,Z 870.218,A -85,B 0,C 180,E1 -3659.34,E2 -3659.34} C_VEL
LIN {X 0,Y 473.788,Z 889.354,A -85,B 0,C 180,E1 -3660.889,E2 -3660.889} C_VEL
LIN {X 0,Y 472.074,Z 907.629,A -85,B 0,C 180,E1 -3662.638,E2 -3662.638} C_VEL
LIN {X 0,Y 470.695,Z 921.182,A -85,B 0,C 180,E1 -3664.185,E2 -3664.185} C_VEL
LIN {X 0,Y 469.011,Z 935.914,A -85,B 0,C 180,E1 -3666.239,E2 -3666.239} C_VEL
LIN {X 0,Y 467.472,Z 950.069,A -85,B 0,C 180,E1 -3668.546,E2 -3668.546} C_VEL
LIN {X 0,Y 466.193,Z 963.106,A -85,B 0,C 180,E1 -3671.053,E2 -3671.053} C_VEL
LIN {X 0,Y 465.25,Z 974.411,A -85,B 0,C 180,E1 -3673.648,E2 -3673.648} C_VEL
LIN {X 0,Y 464.58,Z 984.349,A -85,B 0,C 180,E1 -3676.432,E2 -3676.432} C_VEL
LIN {X 0,Y 464.198,Z 992.209,A -85,B 0,C 180,E1 -3679.199,E2 -3679.199} C_VEL
LIN {X 0,Y 464.007,Z 998.149,A -85,B 0,C 180,E1 -3681.948,E2 -3681.948} C_VEL
LIN {X 0,Y 463.919,Z 1002.133,A -85,B 0,C 180,E1 -3684.558,E2 -3684.558} C_VEL
LIN {X 0,Y 463.897,Z 1004.429,A -85,B 0,C 180,E1 -3687.035,E2 -3687.035} C_VEL
LIN {X 0,Y 463.894,Z 1005.385,A -85,B 0,C 180,E1 -3689.382,E2 -3689.382} C_VEL
LIN {X 0,Y 463.907,Z 1005.052,A -85,B 0,C 180,E1 -3691.976,E2 -3691.976} C_VEL
LIN {X 0,Y 463.913,Z 1002.996,A -85,B 0,C 180,E1 -3694.697,E2 -3694.697} C_VEL
LIN {X 0,Y 463.955,Z 999.439,A -85,B 0,C 180,E1 -3697.305,E2 -3697.305} C_VEL
LIN {X 0,Y 464.1,Z 994.301,A -85,B 0,C 180,E1 -3699.924,E2 -3699.924} C_VEL
LIN {X 0,Y 464.429,Z 987.074,A -85,B 0,C 180,E1 -3702.685,E2 -3702.685} C_VEL
LIN {X 0,Y 465.003,Z 977.809,A -85,B 0,C 180,E1 -3705.463,E2 -3705.463} C_VEL
LIN {X 0,Y 465.913,Z 966.307,A -85,B 0,C 180,E1 -3708.259,E2 -3708.259} C_VEL
LIN {X 0,Y 467.109,Z 953.631,A -85,B 0,C 180,E1 -3710.813,E2 -3710.813} C_VEL
LIN {X 0,Y 468.629,Z 939.294,A -85,B 0,C 180,E1 -3713.248,E2 -3713.248} C_VEL
LIN {X 0,Y 470.477,Z 923.216,A -85,B 0,C 180,E1 -3715.557,E2 -3715.557} C_VEL
LIN {X 0,Y 471.963,Z 908.999,A -85,B 0,C 180,E1 -3717.232,E2 -3717.232} C_VEL
LIN {X 0,Y 473.901,Z 890.053,A -85,B 0,C 180,E1 -3719.135,E2 -3719.135} C_VEL
LIN {X 0,Y 475.892,Z 869.893,A -85,B 0,C 180,E1 -3720.84,E2 -3720.84} C_VEL
LIN {X 0,Y 477.88,Z 848.121,A -85,B 0,C 180,E1 -3722.386,E2 -3722.386} C_VEL
LIN {X 0,Y 479.783,Z 826.105,A -85,B 0,C 180,E1 -3723.665,E2 -3723.665} C_VEL
LIN {X 0,Y 481.405,Z 804.138,A -85,B 0,C 180,E1 -3724.686,E2 -3724.686} C_VEL
LIN {X 0,Y 482.793,Z 781.78,A -85,B 0,C 180,E1 -3725.483,E2 -3725.483} C_VEL
LIN {X 0,Y 483.917,Z 758.946,A -85,B 0,C 180,E1 -3726.076,E2 -3726.076} C_VEL
LIN {X 0,Y 485.103,Z 717.709,A -85,B 0,C 180,E1 -3726.781,E2 -3726.781} C_VEL
LIN {X 0,Y 489.955,Z 701.377,A -85,B 0,C 180,E1 -3727.528,E2 -3727.528} C_VEL
LIN {X 0,Y 496.674,Z 681.71,A -85,B 0,C 180,E1 -3728.319,E2 -3728.319} C_VEL
LIN {X 0,Y 503.7,Z 665.475,A -85,B 0,C 180,E1 -3728.849,E2 -3728.849} C_VEL
LIN {X 0,Y 509.711,Z 650.099,A -85,B 0,C 180,E1 -3729.388,E2 -3729.388} C_VEL
LIN {X 0,Y 518.97,Z 631.509,A -85,B 0,C 180,E1 -3729.908,E2 -3729.908} C_VEL
LIN {X 0,Y 533.457,Z 606.103,A -85,B 0,C 180,E1 -3730.429,E2 -3730.429} C_VEL
LIN {X 0,Y 547.573,Z 582.418,A -85,B 0,C 180,E1 -3730.821,E2 -3730.821} C_VEL
LIN {X 0,Y 550.957,Z 573.933,A -85,B 0,C 180,E1 -3731.083,E2 -3731.083} C_VEL
LIN {X 0,Y 539.246,Z 569.343,A -85,B 0,C 180,E1 -3732.285,E2 -3732.285} C_VEL
LIN {X 0,Y 528.605,Z 563.082,A -85,B 0,C 180,E1 -3733.578,E2 -3733.578} C_VEL
LIN {X 0,Y 519.311,Z 555.237,A -85,B 0,C 180,E1 -3734.959,E2 -3734.959} C_VEL
LIN {X 0,Y 511.587,Z 545.868,A -85,B 0,C 180,E1 -3736.377,E2 -3736.377} C_VEL
LIN {X 0,Y 505.668,Z 535.453,A -85,B 0,C 180,E1 -3737.757,E2 -3737.757} C_VEL
LIN {X 0,Y 501.233,Z 523.739,A -85,B 0,C 180,E1 -3739.134,E2 -3739.134} C_VEL
LIN {X 0,Y 498.302,Z 510.559,A -85,B 0,C 180,E1 -3740.501,E2 -3740.501} C_VEL
LIN {X 0,Y 496.79,Z 493.865,A -85,B 0,C 180,E1 -3742.039,E2 -3742.039} C_VEL
LIN {X 0,Y 497.114,Z 475.716,A -85,B 0,C 180,E1 -3743.509,E2 -3743.509} C_VEL
LIN {X 0,Y 500.666,Z 436.779,A -85,B 0,C 180,E1 -3746.415,E2 -3746.415} C_VEL
LIN {X 0,Y 490.031,Z 417.113,A -85,B 0,C 180,E1 -3749.737,E2 -3749.737} C_VEL
LIN {X 0,Y 481.135,Z 401.562,A -85,B 0,C 180,E1 -3752.661,E2 -3752.661} C_VEL
LIN {X 0,Y 475.553,Z 391.837,A -85,B 0,C 180,E1 -3754.602,E2 -3754.602} C_VEL
LIN {X 0,Y 472.974,Z 387.372,A -85,B 0,C 180,E1 -3755.523,E2 -3755.523} C_VEL
LIN {X 0,Y 470.526,Z 382.855,A -85,B 0,C 180,E1 -3756.454,E2 -3756.454} C_VEL
LIN {X 0,Y 468.227,Z 379.102,A -85,B 0,C 180,E1 -3757.294,E2 -3757.294} C_VEL
LIN {X 0,Y 467.383,Z 377.581,A -85,B 0,C 180,E1 -3757.618,E2 -3757.618} C_VEL
LIN {X 0,Y 465.462,Z 374.616,A -85,B 0,C 180,E1 -3758.317,E2 -3758.317} C_VEL
LIN {X 0,Y 465.013,Z 372.808,A -85,B 0,C 180,E1 -3758.643,E2 -3758.643} C_VEL
LIN {X 0,Y 465.01,Z 372.807,A -85,B 0,C 180,E1 -3762.481,E2 -3762.481} C_VEL
LIN {X 0,Y 464.987,Z 372.811,A -85,B 0,C 180,E1 -3766.065,E2 -3766.065} C_VEL
LIN {X 0,Y 464.994,Z 372.813,A -85,B 0,C 180,E1 -3769.845,E2 -3769.845} C_VEL
LIN {X 0,Y 465.003,Z 372.814,A -85,B 0,C 180,E1 -3773.457,E2 -3773.457} C_VEL
LIN {X 0,Y 464.998,Z 372.817,A -85,B 0,C 180,E1 -3777.166,E2 -3777.166} C_VEL
LIN {X 0,Y 464.998,Z 372.813,A -85,B 0,C 180,E1 -3780.74,E2 -3780.74} C_VEL
LIN {X 0,Y 464.999,Z 372.819,A -85,B 0,C 180,E1 -3784.564,E2 -3784.564} C_VEL
LIN {X 0,Y 464.997,Z 372.816,A -85,B 0,C 180,E1 -3788.159,E2 -3788.159} C_VEL
LIN {X 0,Y 464.984,Z 372.816,A -85,B 0,C 180,E1 -3791.934,E2 -3791.934} C_VEL
LIN {X 0,Y 465.017,Z 372.808,A -85,B 0,C 180,E1 -3795.591,E2 -3795.591} C_VEL
LIN {X 0,Y 465.01,Z 372.815,A -85,B 0,C 180,E1 -3799.338,E2 -3799.338} C_VEL
LIN {X 0,Y 464.995,Z 372.812,A -85,B 0,C 180,E1 -3802.905,E2 -3802.905} C_VEL
LIN {X 0,Y 464.972,Z 372.812,A -85,B 0,C 180,E1 -3806.707,E2 -3806.707} C_VEL
LIN {X 0,Y 465.017,Z 372.81,A -85,B 0,C 180,E1 -3810.351,E2 -3810.351} C_VEL
LIN {X 0,Y 465.008,Z 372.808,A -85,B 0,C 180,E1 -3814.139,E2 -3814.139} C_VEL
LIN {X 0,Y 464.995,Z 372.795,A -85,B 0,C 180,E1 -3817.794,E2 -3817.794} C_VEL
LIN {X 0,Y 464.974,Z 372.798,A -85,B 0,C 180,E1 -3821.555,E2 -3821.555} C_VEL
LIN {X 0,Y 465.01,Z 372.815,A -85,B 0,C 180,E1 -3825.2,E2 -3825.2} C_VEL
LIN {X 0,Y 464.994,Z 372.817,A -85,B 0,C 180,E1 -3828.854,E2 -3828.854} C_VEL
LIN {X 0,Y 465.006,Z 372.841,A -85,B 0,C 180,E1 -3831.186,E2 -3831.186} C_VEL
LIN {X 0,Y 466.368,Z 376.361,A -85,B 0,C 180,E1 -3831.582,E2 -3831.582} C_VEL
LIN {X 0,Y 474.348,Z 395.672,A -85,B 0,C 180,E1 -3833.835,E2 -3833.835} C_VEL
LIN {X 0,Y 479.495,Z 409.627,A -85,B 0,C 180,E1 -3835.408,E2 -3835.408} C_VEL
LIN {X 0,Y 477.539,Z 454.753,A -85,B 0,C 180,E1 -3838.91,E2 -3838.91} C_VEL
LIN {X 0,Y 477.014,Z 475.411,A -85,B 0,C 180,E1 -3840.414,E2 -3840.414} C_VEL
LIN {X 0,Y 476.373,Z 481.482,A -85,B 0,C 180,E1 -3840.728,E2 -3840.728} C_VEL
LIN {X 0,Y 474.483,Z 490.062,A -85,B 0,C 180,E1 -3840.929,E2 -3840.929} C_VEL
LIN {X 0,Y 471.301,Z 504.538,A -85,B 0,C 180,E1 -3841.026,E2 -3841.026} C_VEL
LIN {X 0,Y 470.843,Z 510.2,A -85,B 0,C 180,E1 -3841.092,E2 -3841.092} C_VEL
LIN {X 0,Y 467.991,Z 694.738,A -85,B 0,C 180,E1 -3844.09,E2 -3844.09} C_VEL
LIN {X 0,Y 467.563,Z 713.288,A -85,B 0,C 180,E1 -3844.612,E2 -3844.612} C_VEL
LIN {X 0,Y 466.884,Z 730.665,A -85,B 0,C 180,E1 -3845.317,E2 -3845.317} C_VEL
LIN {X 0,Y 465.954,Z 747.323,A -85,B 0,C 180,E1 -3846.208,E2 -3846.208} C_VEL
LIN {X 0,Y 464.85,Z 763.384,A -85,B 0,C 180,E1 -3847.296,E2 -3847.296} C_VEL
LIN {X 0,Y 463.616,Z 779.233,A -85,B 0,C 180,E1 -3848.625,E2 -3848.625} C_VEL
LIN {X 0,Y 462.332,Z 793.519,A -85,B 0,C 180,E1 -3850.086,E2 -3850.086} C_VEL
LIN {X 0,Y 461.033,Z 807.279,A -85,B 0,C 180,E1 -3851.789,E2 -3851.789} C_VEL
LIN {X 0,Y 459.869,Z 819.255,A -85,B 0,C 180,E1 -3853.582,E2 -3853.582} C_VEL
LIN {X 0,Y 458.807,Z 830.444,A -85,B 0,C 180,E1 -3855.615,E2 -3855.615} C_VEL
LIN {X 0,Y 457.964,Z 840.018,A -85,B 0,C 180,E1 -3857.774,E2 -3857.774} C_VEL
LIN {X 0,Y 457.303,Z 848.019,A -85,B 0,C 180,E1 -3860.054,E2 -3860.054} C_VEL
LIN {X 0,Y 456.888,Z 854.129,A -85,B 0,C 180,E1 -3862.329,E2 -3862.329} C_VEL
LIN {X 0,Y 456.65,Z 858.725,A -85,B 0,C 180,E1 -3864.724,E2 -3864.724} C_VEL
LIN {X 0,Y 456.525,Z 861.574,A -85,B 0,C 180,E1 -3867.113,E2 -3867.113} C_VEL
LIN {X 0,Y 456.481,Z 862.764,A -85,B 0,C 180,E1 -3869.498,E2 -3869.498} C_VEL
LIN {X 0,Y 456.499,Z 862.325,A -85,B 0,C 180,E1 -3871.883,E2 -3871.883} C_VEL
LIN {X 0,Y 456.59,Z 860.245,A -85,B 0,C 180,E1 -3874.27,E2 -3874.27} C_VEL
LIN {X 0,Y 456.762,Z 856.466,A -85,B 0,C 180,E1 -3876.663,E2 -3876.663} C_VEL
LIN {X 0,Y 457.078,Z 851.199,A -85,B 0,C 180,E1 -3878.935,E2 -3878.935} C_VEL
LIN {X 0,Y 457.609,Z 844.144,A -85,B 0,C 180,E1 -3881.214,E2 -3881.214} C_VEL
LIN {X 0,Y 458.339,Z 835.608,A -85,B 0,C 180,E1 -3883.37,E2 -3883.37} C_VEL
LIN {X 0,Y 459.259,Z 825.63,A -85,B 0,C 180,E1 -3885.403,E2 -3885.403} C_VEL
LIN {X 0,Y 460.377,Z 814.201,A -85,B 0,C 180,E1 -3887.31,E2 -3887.31} C_VEL
LIN {X 0,Y 461.616,Z 801.255,A -85,B 0,C 180,E1 -3889.091,E2 -3889.091} C_VEL
LIN {X 0,Y 462.916,Z 787.273,A -85,B 0,C 180,E1 -3890.68,E2 -3890.68} C_VEL
LIN {X 0,Y 464.193,Z 772.356,A -85,B 0,C 180,E1 -3892.078,E2 -3892.078} C_VEL
LIN {X 0,Y 465.341,Z 756.583,A -85,B 0,C 180,E1 -3893.288,E2 -3893.288} C_VEL
LIN {X 0,Y 466.411,Z 739.966,A -85,B 0,C 180,E1 -3894.306,E2 -3894.306} C_VEL
LIN {X 0,Y 467.26,Z 722.165,A -85,B 0,C 180,E1 -3895.147,E2 -3895.147} C_VEL
LIN {X 0,Y 467.818,Z 703.868,A -85,B 0,C 180,E1 -3895.773,E2 -3895.773} C_VEL
LIN {X 0,Y 468.127,Z 683.601,A -85,B 0,C 180,E1 -3896.213,E2 -3896.213} C_VEL
LIN {X 0,Y 470.961,Z 492.643,A -85,B 0,C 180,E1 -3899.296,E2 -3899.296} C_VEL
LIN {X 0,Y 469.957,Z 485.721,A -85,B 0,C 180,E1 -3899.521,E2 -3899.521} C_VEL
LIN {X 0,Y 470.7,Z 454.233,A -85,B 0,C 180,E1 -3901.79,E2 -3901.79} C_VEL
LIN {X 0,Y 472.582,Z 412.616,A -85,B 0,C 180,E1 -3905.036,E2 -3905.036} C_VEL
LIN {X 0,Y 464.663,Z 391.95,A -85,B 0,C 180,E1 -3907.437,E2 -3907.437} C_VEL
LIN {X 0,Y 458.036,Z 376.73,A -85,B 0,C 180,E1 -3909.276,E2 -3909.276} C_VEL
LIN {X 0,Y 457.04,Z 373.799,A -85,B 0,C 180,E1 -3909.64,E2 -3909.64} C_VEL
LIN {X 0,Y 457.073,Z 373.793,A -85,B 0,C 180,E1 -3913.243,E2 -3913.243} C_VEL
LIN {X 0,Y 457.037,Z 373.903,A -85,B 0,C 180,E1 -3916.703,E2 -3916.703} C_VEL
LIN {X 0,Y 458.168,Z 376.973,A -85,B 0,C 180,E1 -3917.16,E2 -3917.16} C_VEL
LIN {X 0,Y 465.146,Z 392.593,A -85,B 0,C 180,E1 -3919.548,E2 -3919.548} C_VEL
LIN {X 0,Y 473.258,Z 412.646,A -85,B 0,C 180,E1 -3922.369,E2 -3922.369} C_VEL
LIN {X 0,Y 475.39,Z 418.753,A -85,B 0,C 180,E1 -3923.171,E2 -3923.171} C_VEL
LIN {X 0,Y 472.383,Z 461.694,A -85,B 0,C 180,E1 -3926.95,E2 -3926.95} C_VEL
LIN {X 0,Y 469.606,Z 504.902,A -85,B 0,C 180,E1 -3930.679,E2 -3930.679} C_VEL
LIN {X 0,Y 466.991,Z 549.064,A -85,B 0,C 180,E1 -3934.442,E2 -3934.442} C_VEL
LIN {X 0,Y 464.661,Z 593.96,A -85,B 0,C 180,E1 -3938.211,E2 -3938.211} C_VEL
LIN {X 0,Y 464.565,Z 598.086,A -85,B 0,C 180,E1 -3938.524,E2 -3938.524} C_VEL
LIN {X 0,Y 465.316,Z 605.899,A -85,B 0,C 180,E1 -3938.727,E2 -3938.727} C_VEL
LIN {X 0,Y 462.358,Z 743.675,A -85,B 0,C 180,E1 -3941.366,E2 -3941.366} C_VEL
LIN {X 0,Y 461.99,Z 760.674,A -85,B 0,C 180,E1 -3941.939,E2 -3941.939} C_VEL
LIN {X 0,Y 461.477,Z 775.611,A -85,B 0,C 180,E1 -3942.667,E2 -3942.667} C_VEL
LIN {X 0,Y 460.785,Z 791.151,A -85,B 0,C 180,E1 -3943.68,E2 -3943.68} C_VEL
LIN {X 0,Y 460.086,Z 804.321,A -85,B 0,C 180,E1 -3944.777,E2 -3944.777} C_VEL
LIN {X 0,Y 459.296,Z 817.966,A -85,B 0,C 180,E1 -3946.209,E2 -3946.209} C_VEL
LIN {X 0,Y 458.626,Z 829.108,A -85,B 0,C 180,E1 -3947.663,E2 -3947.663} C_VEL
LIN {X 0,Y 457.986,Z 839.916,A -85,B 0,C 180,E1 -3949.433,E2 -3949.433} C_VEL
LIN {X 0,Y 457.518,Z 848.457,A -85,B 0,C 180,E1 -3951.2,E2 -3951.2} C_VEL
LIN {X 0,Y 457.16,Z 855.914,A -85,B 0,C 180,E1 -3953.217,E2 -3953.217} C_VEL
LIN {X 0,Y 456.956,Z 861.029,A -85,B 0,C 180,E1 -3955.104,E2 -3955.104} C_VEL
LIN {X 0,Y 456.867,Z 864.83,A -85,B 0,C 180,E1 -3957.24,E2 -3957.24} C_VEL
LIN {X 0,Y 456.855,Z 866.672,A -85,B 0,C 180,E1 -3959.247,E2 -3959.247} C_VEL
LIN {X 0,Y 456.929,Z 866.764,A -85,B 0,C 180,E1 -3961.379,E2 -3961.379} C_VEL
LIN {X 0,Y 457.062,Z 865.178,A -85,B 0,C 180,E1 -3963.386,E2 -3963.386} C_VEL
LIN {X 0,Y 457.327,Z 861.57,A -85,B 0,C 180,E1 -3965.52,E2 -3965.52} C_VEL
LIN {X 0,Y 457.691,Z 856.674,A -85,B 0,C 180,E1 -3967.405,E2 -3967.405} C_VEL
LIN {X 0,Y 458.259,Z 849.402,A -85,B 0,C 180,E1 -3969.418,E2 -3969.418} C_VEL
LIN {X 0,Y 458.901,Z 841.032,A -85,B 0,C 180,E1 -3971.181,E2 -3971.181} C_VEL
LIN {X 0,Y 459.661,Z 831.202,A -85,B 0,C 180,E1 -3972.819,E2 -3972.819} C_VEL
LIN {X 0,Y 460.478,Z 820.328,A -85,B 0,C 180,E1 -3974.267,E2 -3974.267} C_VEL
LIN {X 0,Y 461.365,Z 807.294,A -85,B 0,C 180,E1 -3975.653,E2 -3975.653} C_VEL
LIN {X 0,Y 462.142,Z 793.751,A -85,B 0,C 180,E1 -3976.788,E2 -3976.788} C_VEL
LIN {X 0,Y 462.796,Z 779.228,A -85,B 0,C 180,E1 -3977.735,E2 -3977.735} C_VEL
LIN {X 0,Y 463.261,Z 763.648,A -85,B 0,C 180,E1 -3978.481,E2 -3978.481} C_VEL
LIN {X 0,Y 463.514,Z 747.465,A -85,B 0,C 180,E1 -3979.013,E2 -3979.013} C_VEL
LIN {X 0,Y 465.574,Z 697.788,A -85,B 0,C 180,E1 -3980.285,E2 -3980.285} C_VEL
LIN {X 0,Y 470.889,Z 617.874,A -85,B 0,C 180,E1 -3982.437,E2 -3982.437} C_VEL
LIN {X 0,Y 473.632,Z 609.456,A -85,B 0,C 180,E1 -3983.012,E2 -3983.012} C_VEL
LIN {X 0,Y 479.577,Z 568.894,A -85,B 0,C 180,E1 -3986.966,E2 -3986.966} C_VEL
LIN {X 0,Y 486.159,Z 536.589,A -85,B 0,C 180,E1 -3990.325,E2 -3990.325} C_VEL
LIN {X 0,Y 492.711,Z 513.729,A -85,B 0,C 180,E1 -3992.87,E2 -3992.87} C_VEL
LIN {X 0,Y 499.945,Z 495.691,A -85,B 0,C 180,E1 -3995.028,E2 -3995.028} C_VEL
LIN {X 0,Y 503.084,Z 489.535,A -85,B 0,C 180,E1 -3995.817,E2 -3995.817} C_VEL
LIN {X 0,Y 497.345,Z 498.984,A -85,B 0,C 180,E1 -3997.093,E2 -3997.093} C_VEL
LIN {X 0,Y 493.624,Z 508.567,A -85,B 0,C 180,E1 -3998.45,E2 -3998.45} C_VEL
LIN {X 0,Y 492.101,Z 517.899,A -85,B 0,C 180,E1 -3999.793,E2 -3999.793} C_VEL
LIN {X 0,Y 492.665,Z 527.292,A -85,B 0,C 180,E1 -4001.154,E2 -4001.154} C_VEL
LIN {X 0,Y 495.464,Z 536.947,A -85,B 0,C 180,E1 -4002.559,E2 -4002.559} C_VEL
LIN {X 0,Y 500.302,Z 546.196,A -85,B 0,C 180,E1 -4003.906,E2 -4003.906} C_VEL
LIN {X 0,Y 507.822,Z 555.721,A -85,B 0,C 180,E1 -4005.298,E2 -4005.298} C_VEL
LIN {X 0,Y 516.78,Z 563.898,A -85,B 0,C 180,E1 -4006.514,E2 -4006.514} C_VEL
LIN {X 0,Y 527.633,Z 571.353,A -85,B 0,C 180,E1 -4007.65,E2 -4007.65} C_VEL
LIN {X 0,Y 540.347,Z 577.866,A -85,B 0,C 180,E1 -4008.699,E2 -4008.699} C_VEL
LIN {X 0,Y 541.173,Z 578.339,A -85,B 0,C 180,E1 -4008.768,E2 -4008.768} C_VEL
LIN {X 0,Y 538.951,Z 582.32,A -85,B 0,C 180,E1 -4008.869,E2 -4008.869} C_VEL
LIN {X 0,Y 514.899,Z 620.917,A -85,B 0,C 180,E1 -4009.742,E2 -4009.742} C_VEL
LIN {X 0,Y 504.086,Z 640.949,A -85,B 0,C 180,E1 -4010.305,E2 -4010.305} C_VEL
LIN {X 0,Y 496.804,Z 657.61,A -85,B 0,C 180,E1 -4010.88,E2 -4010.88} C_VEL
LIN {X 0,Y 493.724,Z 665.676,A -85,B 0,C 180,E1 -4011.187,E2 -4011.187} C_VEL
LIN {X 0,Y 486.846,Z 681.347,A -85,B 0,C 180,E1 -4011.741,E2 -4011.741} C_VEL
LIN {X 0,Y 478.067,Z 708.3,A -85,B 0,C 180,E1 -4012.887,E2 -4012.887} C_VEL
LIN {X 0,Y 476.552,Z 714.492,A -85,B 0,C 180,E1 -4013.143,E2 -4013.143} C_VEL
LIN {X 0,Y 475.81,Z 726.944,A -85,B 0,C 180,E1 -4013.317,E2 -4013.317} C_VEL
LIN {X 0,Y 475.064,Z 760.071,A -85,B 0,C 180,E1 -4013.905,E2 -4013.905} C_VEL
LIN {X 0,Y 473.977,Z 783.555,A -85,B 0,C 180,E1 -4014.531,E2 -4014.531} C_VEL
LIN {X 0,Y 472.622,Z 806.591,A -85,B 0,C 180,E1 -4015.381,E2 -4015.381} C_VEL
LIN {X 0,Y 471.129,Z 828.94,A -85,B 0,C 180,E1 -4016.437,E2 -4016.437} C_VEL
LIN {X 0,Y 469.431,Z 850.353,A -85,B 0,C 180,E1 -4017.682,E2 -4017.682} C_VEL
LIN {X 0,Y 467.699,Z 870.96,A -85,B 0,C 180,E1 -4019.13,E2 -4019.13} C_VEL
LIN {X 0,Y 465.878,Z 890.513,A -85,B 0,C 180,E1 -4020.774,E2 -4020.774} C_VEL
LIN {X 0,Y 463.995,Z 909.776,A -85,B 0,C 180,E1 -4022.677,E2 -4022.677} C_VEL
LIN {X 0,Y 462.155,Z 928.048,A -85,B 0,C 180,E1 -4024.826,E2 -4024.826} C_VEL
LIN {X 0,Y 460.843,Z 940.782,A -85,B 0,C 180,E1 -4026.606,E2 -4026.606} C_VEL
LIN {X 0,Y 459.409,Z 953.627,A -85,B 0,C 180,E1 -4028.821,E2 -4028.821} C_VEL
LIN {X 0,Y 458.055,Z 966.884,A -85,B 0,C 180,E1 -4031.548,E2 -4031.548} C_VEL
LIN {X 0,Y 457.113,Z 977.812,A -85,B 0,C 180,E1 -4034.262,E2 -4034.262} C_VEL
LIN {X 0,Y 456.487,Z 987.075,A -85,B 0,C 180,E1 -4037.09,E2 -4037.09} C_VEL
LIN {X 0,Y 456.126,Z 994.296,A -85,B 0,C 180,E1 -4039.9,E2 -4039.9} C_VEL
LIN {X 0,Y 455.962,Z 999.438,A -85,B 0,C 180,E1 -4042.566,E2 -4042.566} C_VEL
LIN {X 0,Y 455.911,Z 1002.997,A -85,B 0,C 180,E1 -4045.219,E2 -4045.219} C_VEL
LIN {X 0,Y 455.904,Z 1005.108,A -85,B 0,C 180,E1 -4048.114,E2 -4048.114} C_VEL
LIN {X 0,Y 455.9,Z 1005.402,A -85,B 0,C 180,E1 -4050.879,E2 -4050.879} C_VEL
LIN {X 0,Y 455.913,Z 1004.032,A -85,B 0,C 180,E1 -4053.646,E2 -4053.646} C_VEL
LIN {X 0,Y 455.951,Z 1001.165,A -85,B 0,C 180,E1 -4056.295,E2 -4056.295} C_VEL
LIN {X 0,Y 456.063,Z 996.461,A -85,B 0,C 180,E1 -4059.082,E2 -4059.082} C_VEL
LIN {X 0,Y 456.325,Z 989.93,A -85,B 0,C 180,E1 -4061.886,E2 -4061.886} C_VEL
LIN {X 0,Y 456.835,Z 981.423,A -85,B 0,C 180,E1 -4064.707,E2 -4064.707} C_VEL
LIN {X 0,Y 457.643,Z 971.29,A -85,B 0,C 180,E1 -4067.416,E2 -4067.416} C_VEL
LIN {X 0,Y 458.766,Z 959.596,A -85,B 0,C 180,E1 -4070.009,E2 -4070.009} C_VEL
LIN {X 0,Y 460.127,Z 947.115,A -85,B 0,C 180,E1 -4072.35,E2 -4072.35} C_VEL
LIN {X 0,Y 461.409,Z 935.494,A -85,B 0,C 180,E1 -4074.177,E2 -4074.177} C_VEL
LIN {X 0,Y 463.106,Z 919.666,A -85,B 0,C 180,E1 -4076.27,E2 -4076.27} C_VEL
LIN {X 0,Y 464.972,Z 902.38,A -85,B 0,C 180,E1 -4078.234,E2 -4078.234} C_VEL
LIN {X 0,Y 467.096,Z 882.642,A -85,B 0,C 180,E1 -4080.141,E2 -4080.141} C_VEL
LIN {X 0,Y 469.138,Z 862.773,A -85,B 0,C 180,E1 -4081.764,E2 -4081.764} C_VEL
LIN {X 0,Y 471.173,Z 841.749,A -85,B 0,C 180,E1 -4083.195,E2 -4083.195} C_VEL
LIN {X 0,Y 473.087,Z 819.604,A -85,B 0,C 180,E1 -4084.427,E2 -4084.427} C_VEL
LIN {X 0,Y 474.829,Z 797.17,A -85,B 0,C 180,E1 -4085.422,E2 -4085.422} C_VEL
LIN {X 0,Y 476.274,Z 774.171,A -85,B 0,C 180,E1 -4086.192,E2 -4086.192} C_VEL
LIN {X 0,Y 477.369,Z 750.523,A -85,B 0,C 180,E1 -4086.735,E2 -4086.735} C_VEL
LIN {X 0,Y 478.366,Z 717.105,A -85,B 0,C 180,E1 -4087.292,E2 -4087.292} C_VEL
LIN {X 0,Y 483.375,Z 700.522,A -85,B 0,C 180,E1 -4088.054,E2 -4088.054} C_VEL
LIN {X 0,Y 490.138,Z 680.997,A -85,B 0,C 180,E1 -4088.85,E2 -4088.85} C_VEL
LIN {X 0,Y 497.214,Z 664.765,A -85,B 0,C 180,E1 -4089.379,E2 -4089.379} C_VEL
LIN {X 0,Y 503.25,Z 649.446,A -85,B 0,C 180,E1 -4089.924,E2 -4089.924} C_VEL
LIN {X 0,Y 512.384,Z 631.012,A -85,B 0,C 180,E1 -4090.445,E2 -4090.445} C_VEL
LIN {X 0,Y 526.689,Z 605.923,A -85,B 0,C 180,E1 -4090.965,E2 -4090.965} C_VEL
LIN {X 0,Y 542.026,Z 579.927,A -85,B 0,C 180,E1 -4091.4,E2 -4091.4} C_VEL
LIN {X 0,Y 542.16,Z 579.155,A -85,B 0,C 180,E1 -4091.438,E2 -4091.438} C_VEL
LIN {X 0,Y 530.284,Z 573.607,A -85,B 0,C 180,E1 -4092.748,E2 -4092.748} C_VEL
LIN {X 0,Y 519.706,Z 566.363,A -85,B 0,C 180,E1 -4094.143,E2 -4094.143} C_VEL
LIN {X 0,Y 511.629,Z 558.625,A -85,B 0,C 180,E1 -4095.446,E2 -4095.446} C_VEL
LIN {X 0,Y 503.987,Z 548.347,A -85,B 0,C 180,E1 -4096.964,E2 -4096.964} C_VEL
LIN {X 0,Y 498.011,Z 536.355,A -85,B 0,C 180,E1 -4098.506,E2 -4098.506} C_VEL
LIN {X 0,Y 494.005,Z 523.731,A -85,B 0,C 180,E1 -4099.938,E2 -4099.938} C_VEL
LIN {X 0,Y 491.578,Z 509.661,A -85,B 0,C 180,E1 -4101.36,E2 -4101.36} C_VEL
LIN {X 0,Y 490.602,Z 492.524,A -85,B 0,C 180,E1 -4102.897,E2 -4102.897} C_VEL
LIN {X 0,Y 491.596,Z 472.44,A -85,B 0,C 180,E1 -4104.495,E2 -4104.495} C_VEL
LIN {X 0,Y 494.643,Z 441.062,A -85,B 0,C 180,E1 -4106.854,E2 -4106.854} C_VEL
LIN {X 0,Y 484.206,Z 421.919,A -85,B 0,C 180,E1 -4110.156,E2 -4110.156} C_VEL
LIN {X 0,Y 476.384,Z 407.979,A -85,B 0,C 180,E1 -4112.771,E2 -4112.771} C_VEL
LIN {X 0,Y 468.227,Z 393.71,A -85,B 0,C 180,E1 -4115.661,E2 -4115.661} C_VEL
LIN {X 0,Y 465.058,Z 388.341,A -85,B 0,C 180,E1 -4116.831,E2 -4116.831} C_VEL
LIN {X 0,Y 462.628,Z 383.903,A -85,B 0,C 180,E1 -4117.777,E2 -4117.777} C_VEL
LIN {X 0,Y 460.43,Z 380.388,A -85,B 0,C 180,E1 -4118.604,E2 -4118.604} C_VEL
LIN {X 0,Y 459.587,Z 378.711,A -85,B 0,C 180,E1 -4118.964,E2 -4118.964} C_VEL
LIN {X 0,Y 457.6,Z 375.931,A -85,B 0,C 180,E1 -4119.671,E2 -4119.671} C_VEL
LIN {X 0,Y 457.045,Z 373.803,A -85,B 0,C 180,E1 -4120.046,E2 -4120.046} C_VEL
LIN {X 0,Y 457.072,Z 373.799,A -85,B 0,C 180,E1 -4123.74,E2 -4123.74} C_VEL
LIN {X 0,Y 457.034,Z 373.806,A -85,B 0,C 180,E1 -4127.363,E2 -4127.363} C_VEL
LIN {X 0,Y 457.066,Z 373.802,A -85,B 0,C 180,E1 -4131.065,E2 -4131.065} C_VEL
LIN {X 0,Y 457.054,Z 373.802,A -85,B 0,C 180,E1 -4134.603,E2 -4134.603} C_VEL
LIN {X 0,Y 457.074,Z 373.801,A -85,B 0,C 180,E1 -4138.371,E2 -4138.371} C_VEL
LIN {X 0,Y 457.033,Z 373.81,A -85,B 0,C 180,E1 -4142.006,E2 -4142.006} C_VEL
LIN {X 0,Y 457.06,Z 373.803,A -85,B 0,C 180,E1 -4145.902,E2 -4145.902} C_VEL
LIN {X 0,Y 457.066,Z 373.803,A -85,B 0,C 180,E1 -4149.57,E2 -4149.57} C_VEL
LIN {X 0,Y 457.079,Z 373.8,A -85,B 0,C 180,E1 -4153.279,E2 -4153.279} C_VEL
LIN {X 0,Y 457.034,Z 373.805,A -85,B 0,C 180,E1 -4156.916,E2 -4156.916} C_VEL
LIN {X 0,Y 457.06,Z 373.801,A -85,B 0,C 180,E1 -4160.622,E2 -4160.622} C_VEL
LIN {X 0,Y 457.067,Z 373.799,A -85,B 0,C 180,E1 -4164.188,E2 -4164.188} C_VEL
LIN {X 0,Y 457.071,Z 373.796,A -85,B 0,C 180,E1 -4168.055,E2 -4168.055} C_VEL
LIN {X 0,Y 457.049,Z 373.795,A -85,B 0,C 180,E1 -4171.671,E2 -4171.671} C_VEL
LIN {X 0,Y 457.057,Z 373.78,A -85,B 0,C 180,E1 -4175.316,E2 -4175.316} C_VEL
LIN {X 0,Y 457.06,Z 373.799,A -85,B 0,C 180,E1 -4178.891,E2 -4178.891} C_VEL
LIN {X 0,Y 457.065,Z 373.776,A -85,B 0,C 180,E1 -4182.529,E2 -4182.529} C_VEL
LIN {X 0,Y 457.051,Z 373.794,A -85,B 0,C 180,E1 -4186.094,E2 -4186.094} C_VEL
LIN {X 0,Y 457.05,Z 373.803,A -85,B 0,C 180,E1 -4189.808,E2 -4189.808} C_VEL
LIN {X 0,Y 457.084,Z 373.817,A -85,B 0,C 180,E1 -4190.507,E2 -4190.507} C_VEL
LIN {X 0,Y 457.974,Z 376.604,A -85,B 0,C 180,E1 -4190.81,E2 -4190.81} C_VEL
LIN {X 0,Y 464.58,Z 391.707,A -85,B 0,C 180,E1 -4192.634,E2 -4192.634} C_VEL
LIN {X 0,Y 472.538,Z 412.808,A -85,B 0,C 180,E1 -4195.078,E2 -4195.078} C_VEL
LIN {X 0,Y 470.575,Z 457.625,A -85,B 0,C 180,E1 -4198.559,E2 -4198.559} C_VEL
LIN {X 0,Y 469.971,Z 486.535,A -85,B 0,C 180,E1 -4200.62,E2 -4200.62} C_VEL
LIN {X 0,Y 471.094,Z 495.221,A -85,B 0,C 180,E1 -4200.85,E2 -4200.85} C_VEL
LIN {X 0,Y 470.843,Z 510.2,A -85,B 0,C 180,E1 -4201.092,E2 -4201.092} C_VEL
LIN {X 0,Y 469.846,Z 517.885,A -85,B 0,C 180,E1 -4201.155,E2 -4201.155} C_VEL
LIN {X 0,Y 464.05,Z 538.327,A -85,B 0,C 180,E1 -4201.103,E2 -4201.103} C_VEL
LIN {X 0,Y 463.286,Z 544.923,A -85,B 0,C 180,E1 -4201.164,E2 -4201.164} C_VEL
LIN {X 0,Y 460.864,Z 695.882,A -85,B 0,C 180,E1 -4203.659,E2 -4203.659} C_VEL
LIN {X 0,Y 460.419,Z 714.5,A -85,B 0,C 180,E1 -4204.189,E2 -4204.189} C_VEL
LIN {X 0,Y 459.708,Z 731.895,A -85,B 0,C 180,E1 -4204.905,E2 -4204.905} C_VEL
LIN {X 0,Y 458.691,Z 749.206,A -85,B 0,C 180,E1 -4205.849,E2 -4205.849} C_VEL
LIN {X 0,Y 457.514,Z 765.402,A -85,B 0,C 180,E1 -4206.972,E2 -4206.972} C_VEL
LIN {X 0,Y 456.213,Z 781.104,A -85,B 0,C 180,E1 -4208.321,E2 -4208.321} C_VEL
LIN {X 0,Y 454.837,Z 795.516,A -85,B 0,C 180,E1 -4209.83,E2 -4209.83} C_VEL
LIN {X 0,Y 453.512,Z 808.639,A -85,B 0,C 180,E1 -4211.49,E2 -4211.49} C_VEL
LIN {X 0,Y 452.202,Z 821.308,A -85,B 0,C 180,E1 -4213.428,E2 -4213.428} C_VEL
LIN {X 0,Y 451.07,Z 832.316,A -85,B 0,C 180,E1 -4215.494,E2 -4215.494} C_VEL
LIN {X 0,Y 450.17,Z 841.765,A -85,B 0,C 180,E1 -4217.689,E2 -4217.689} C_VEL
LIN {X 0,Y 449.502,Z 849.285,A -85,B 0,C 180,E1 -4219.879,E2 -4219.879} C_VEL
LIN {X 0,Y 449.032,Z 855.536,A -85,B 0,C 180,E1 -4222.258,E2 -4222.258} C_VEL
LIN {X 0,Y 448.773,Z 859.99,A -85,B 0,C 180,E1 -4224.631,E2 -4224.631} C_VEL
LIN {X 0,Y 448.632,Z 862.838,A -85,B 0,C 180,E1 -4227.062,E2 -4227.062} C_VEL
LIN {X 0,Y 448.581,Z 864.027,A -85,B 0,C 180,E1 -4229.49,E2 -4229.49} C_VEL
LIN {X 0,Y 448.602,Z 863.588,A -85,B 0,C 180,E1 -4231.916,E2 -4231.916} C_VEL
LIN {X 0,Y 448.705,Z 861.508,A -85,B 0,C 180,E1 -4234.345,E2 -4234.345} C_VEL
LIN {X 0,Y 448.901,Z 857.729,A -85,B 0,C 180,E1 -4236.78,E2 -4236.78} C_VEL
LIN {X 0,Y 449.255,Z 852.461,A -85,B 0,C 180,E1 -4239.092,E2 -4239.092} C_VEL
LIN {X 0,Y 449.841,Z 845.384,A -85,B 0,C 180,E1 -4241.416,E2 -4241.416} C_VEL
LIN {X 0,Y 450.644,Z 836.729,A -85,B 0,C 180,E1 -4243.637,E2 -4243.637} C_VEL
LIN {X 0,Y 451.692,Z 826.178,A -85,B 0,C 180,E1 -4245.8,E2 -4245.8} C_VEL
LIN {X 0,Y 452.905,Z 814.581,A -85,B 0,C 180,E1 -4247.738,E2 -4247.738} C_VEL
LIN {X 0,Y 454.192,Z 801.977,A -85,B 0,C 180,E1 -4249.482,E2 -4249.482} C_VEL
LIN {X 0,Y 455.58,Z 787.882,A -85,B 0,C 180,E1 -4251.096,E2 -4251.096} C_VEL
LIN {X 0,Y 456.934,Z 772.821,A -85,B 0,C 180,E1 -4252.516,E2 -4252.516} C_VEL
LIN {X 0,Y 458.159,Z 756.854,A -85,B 0,C 180,E1 -4253.744,E2 -4253.744} C_VEL
LIN {X 0,Y 459.302,Z 739.523,A -85,B 0,C 180,E1 -4254.8,E2 -4254.8} C_VEL
LIN {X 0,Y 460.198,Z 720.973,A -85,B 0,C 180,E1 -4255.661,E2 -4255.661} C_VEL
LIN {X 0,Y 460.749,Z 702.321,A -85,B 0,C 180,E1 -4256.276,E2 -4256.276} C_VEL
LIN {X 0,Y 461.036,Z 681.065,A -85,B 0,C 180,E1 -4256.71,E2 -4256.71} C_VEL
LIN {X 0,Y 464.045,Z 493.897,A -85,B 0,C 180,E1 -4259.773,E2 -4259.773} C_VEL
LIN {X 0,Y 463.043,Z 487.346,A -85,B 0,C 180,E1 -4259.975,E2 -4259.975} C_VEL
LIN {X 0,Y 463.805,Z 455.878,A -85,B 0,C 180,E1 -4262.246,E2 -4262.246} C_VEL
LIN {X 0,Y 465.662,Z 415.795,A -85,B 0,C 180,E1 -4265.381,E2 -4265.381} C_VEL
LIN {X 0,Y 457.942,Z 395.482,A -85,B 0,C 180,E1 -4267.778,E2 -4267.778} C_VEL
LIN {X 0,Y 450.373,Z 378.242,A -85,B 0,C 180,E1 -4269.912,E2 -4269.912} C_VEL
LIN {X 0,Y 449.081,Z 374.781,A -85,B 0,C 180,E1 -4270.342,E2 -4270.342} C_VEL
LIN {X 0,Y 449.085,Z 374.777,A -85,B 0,C 180,E1 -4274.016,E2 -4274.016} C_VEL
LIN {X 0,Y 449.115,Z 374.912,A -85,B 0,C 180,E1 -4275.855,E2 -4275.855} C_VEL
LIN {X 0,Y 450.361,Z 378.247,A -85,B 0,C 180,E1 -4276.366,E2 -4276.366} C_VEL
LIN {X 0,Y 456.472,Z 391.777,A -85,B 0,C 180,E1 -4278.515,E2 -4278.515} C_VEL
LIN {X 0,Y 464.227,Z 410.353,A -85,B 0,C 180,E1 -4281.232,E2 -4281.232} C_VEL
LIN {X 0,Y 468.575,Z 421.908,A -85,B 0,C 180,E1 -4282.809,E2 -4282.809} C_VEL
LIN {X 0,Y 465.444,Z 464.191,A -85,B 0,C 180,E1 -4286.563,E2 -4286.563} C_VEL
LIN {X 0,Y 462.472,Z 507.658,A -85,B 0,C 180,E1 -4290.357,E2 -4290.357} C_VEL
LIN {X 0,Y 459.738,Z 551.743,A -85,B 0,C 180,E1 -4294.147,E2 -4294.147} C_VEL
LIN {X 0,Y 457.244,Z 597.11,A -85,B 0,C 180,E1 -4297.998,E2 -4297.998} C_VEL
LIN {X 0,Y 457.31,Z 599.233,A -85,B 0,C 180,E1 -4298.124,E2 -4298.124} C_VEL
LIN {X 0,Y 458.027,Z 606.857,A -85,B 0,C 180,E1 -4298.327,E2 -4298.327} C_VEL
LIN {X 0,Y 454.812,Z 744.433,A -85,B 0,C 180,E1 -4301.045,E2 -4301.045} C_VEL
LIN {X 0,Y 454.419,Z 761.627,A -85,B 0,C 180,E1 -4301.635,E2 -4301.635} C_VEL
LIN {X 0,Y 453.832,Z 777.508,A -85,B 0,C 180,E1 -4302.432,E2 -4302.432} C_VEL
LIN {X 0,Y 453.114,Z 792.869,A -85,B 0,C 180,E1 -4303.461,E2 -4303.461} C_VEL
LIN {X 0,Y 452.311,Z 806.975,A -85,B 0,C 180,E1 -4304.683,E2 -4304.683} C_VEL
LIN {X 0,Y 451.518,Z 820.024,A -85,B 0,C 180,E1 -4306.097,E2 -4306.097} C_VEL
LIN {X 0,Y 450.815,Z 830.974,A -85,B 0,C 180,E1 -4307.576,E2 -4307.576} C_VEL
LIN {X 0,Y 450.149,Z 841.695,A -85,B 0,C 180,E1 -4309.376,E2 -4309.376} C_VEL
LIN {X 0,Y 449.655,Z 850.117,A -85,B 0,C 180,E1 -4311.174,E2 -4311.174} C_VEL
LIN {X 0,Y 449.285,Z 857.524,A -85,B 0,C 180,E1 -4313.226,E2 -4313.226} C_VEL
LIN {X 0,Y 449.056,Z 862.814,A -85,B 0,C 180,E1 -4315.274,E2 -4315.274} C_VEL
LIN {X 0,Y 448.982,Z 866.313,A -85,B 0,C 180,E1 -4317.319,E2 -4317.319} C_VEL
LIN {X 0,Y 448.971,Z 868.075,A -85,B 0,C 180,E1 -4319.362,E2 -4319.362} C_VEL
LIN {X 0,Y 449.066,Z 868.137,A -85,B 0,C 180,E1 -4321.531,E2 -4321.531} C_VEL
LIN {X 0,Y 449.216,Z 866.458,A -85,B 0,C 180,E1 -4323.573,E2 -4323.573} C_VEL
LIN {X 0,Y 449.53,Z 862.814,A -85,B 0,C 180,E1 -4325.744,E2 -4325.744} C_VEL
LIN {X 0,Y 449.964,Z 857.418,A -85,B 0,C 180,E1 -4327.79,E2 -4327.79} C_VEL
LIN {X 0,Y 450.582,Z 850.513,A -85,B 0,C 180,E1 -4329.709,E2 -4329.709} C_VEL
LIN {X 0,Y 451.284,Z 842.028,A -85,B 0,C 180,E1 -4331.502,E2 -4331.502} C_VEL
LIN {X 0,Y 452.125,Z 832.122,A -85,B 0,C 180,E1 -4333.166,E2 -4333.166} C_VEL
LIN {X 0,Y 453.053,Z 820.569,A -85,B 0,C 180,E1 -4334.702,E2 -4334.702} C_VEL
LIN {X 0,Y 453.976,Z 807.984,A -85,B 0,C 180,E1 -4336.046,E2 -4336.046} C_VEL
LIN {X 0,Y 454.804,Z 794.229,A -85,B 0,C 180,E1 -4337.199,E2 -4337.199} C_VEL
LIN {X 0,Y 455.457,Z 780.715,A -85,B 0,C 180,E1 -4338.09,E2 -4338.09} C_VEL
LIN {X 0,Y 455.974,Z 764.746,A -85,B 0,C 180,E1 -4338.871,E2 -4338.871} C_VEL
LIN {X 0,Y 456.24,Z 748.982,A -85,B 0,C 180,E1 -4339.399,E2 -4339.399} C_VEL
LIN {X 0,Y 458.333,Z 703.801,A -85,B 0,C 180,E1 -4340.63,E2 -4340.63} C_VEL
LIN {X 0,Y 464.521,Z 620.424,A -85,B 0,C 180,E1 -4342.996,E2 -4342.996} C_VEL
LIN {X 0,Y 467.613,Z 611.184,A -85,B 0,C 180,E1 -4343.635,E2 -4343.635} C_VEL
LIN {X 0,Y 473.795,Z 572.769,A -85,B 0,C 180,E1 -4347.458,E2 -4347.458} C_VEL
LIN {X 0,Y 480.77,Z 541.61,A -85,B 0,C 180,E1 -4350.771,E2 -4350.771} C_VEL
LIN {X 0,Y 487.479,Z 520.225,A -85,B 0,C 180,E1 -4353.205,E2 -4353.205} C_VEL
LIN {X 0,Y 494.917,Z 503.095,A -85,B 0,C 180,E1 -4355.295,E2 -4355.295} C_VEL
LIN {X 0,Y 496.942,Z 499.297,A -85,B 0,C 180,E1 -4355.821,E2 -4355.821} C_VEL
LIN {X 0,Y 491.433,Z 508.662,A -85,B 0,C 180,E1 -4357.176,E2 -4357.176} C_VEL
LIN {X 0,Y 488.077,Z 518.106,A -85,B 0,C 180,E1 -4358.599,E2 -4358.599} C_VEL
LIN {X 0,Y 487.019,Z 527.42,A -85,B 0,C 180,E1 -4360.023,E2 -4360.023} C_VEL
LIN {X 0,Y 488.171,Z 536.672,A -85,B 0,C 180,E1 -4361.441,E2 -4361.441} C_VEL
LIN {X 0,Y 491.751,Z 546.443,A -85,B 0,C 180,E1 -4362.933,E2 -4362.933} C_VEL
LIN {X 0,Y 497.193,Z 555.306,A -85,B 0,C 180,E1 -4364.281,E2 -4364.281} C_VEL
LIN {X 0,Y 504.938,Z 564.191,A -85,B 0,C 180,E1 -4365.629,E2 -4365.629} C_VEL
LIN {X 0,Y 514.84,Z 572.454,A -85,B 0,C 180,E1 -4366.904,E2 -4366.904} C_VEL
LIN {X 0,Y 525.953,Z 579.503,A -85,B 0,C 180,E1 -4368.013,E2 -4368.013} C_VEL
LIN {X 0,Y 531.065,Z 582.32,A -85,B 0,C 180,E1 -4368.455,E2 -4368.455} C_VEL
LIN {X 0,Y 508.61,Z 618.533,A -85,B 0,C 180,E1 -4369.256,E2 -4369.256} C_VEL
LIN {X 0,Y 497.514,Z 639.151,A -85,B 0,C 180,E1 -4369.825,E2 -4369.825} C_VEL
LIN {X 0,Y 490.019,Z 656.276,A -85,B 0,C 180,E1 -4370.413,E2 -4370.413} C_VEL
LIN {X 0,Y 487.067,Z 663.975,A -85,B 0,C 180,E1 -4370.706,E2 -4370.706} C_VEL
LIN {X 0,Y 480.143,Z 679.683,A -85,B 0,C 180,E1 -4371.261,E2 -4371.261} C_VEL
LIN {X 0,Y 470.928,Z 707.693,A -85,B 0,C 180,E1 -4372.457,E2 -4372.457} C_VEL
LIN {X 0,Y 469.653,Z 712.959,A -85,B 0,C 180,E1 -4372.672,E2 -4372.672} C_VEL
LIN {X 0,Y 468.728,Z 725.853,A -85,B 0,C 180,E1 -4372.849,E2 -4372.849} C_VEL
LIN {X 0,Y 467.886,Z 758.996,A -85,B 0,C 180,E1 -4373.459,E2 -4373.459} C_VEL
LIN {X 0,Y 466.682,Z 782.757,A -85,B 0,C 180,E1 -4374.116,E2 -4374.116} C_VEL
LIN {X 0,Y 465.229,Z 805.71,A -85,B 0,C 180,E1 -4374.982,E2 -4374.982} C_VEL
LIN {X 0,Y 463.612,Z 828.562,A -85,B 0,C 180,E1 -4376.083,E2 -4376.083} C_VEL
LIN {X 0,Y 461.804,Z 850.352,A -85,B 0,C 180,E1 -4377.376,E2 -4377.376} C_VEL
LIN {X 0,Y 459.997,Z 870.703,A -85,B 0,C 180,E1 -4378.847,E2 -4378.847} C_VEL
LIN {X 0,Y 458.17,Z 889.474,A -85,B 0,C 180,E1 -4380.449,E2 -4380.449} C_VEL
LIN {X 0,Y 456.295,Z 908.207,A -85,B 0,C 180,E1 -4382.319,E2 -4382.319} C_VEL
LIN {X 0,Y 454.419,Z 926.211,A -85,B 0,C 180,E1 -4384.452,E2 -4384.452} C_VEL
LIN {X 0,Y 452.66,Z 943.24,A -85,B 0,C 180,E1 -4386.847,E2 -4386.847} C_VEL
LIN {X 0,Y 451.293,Z 956.713,A -85,B 0,C 180,E1 -4389.102,E2 -4389.102} C_VEL
LIN {X 0,Y 450.314,Z 966.303,A -85,B 0,C 180,E1 -4391.084,E2 -4391.084} C_VEL
LIN {X 0,Y 449.272,Z 977.334,A -85,B 0,C 180,E1 -4393.847,E2 -4393.847} C_VEL
LIN {X 0,Y 448.594,Z 986.3,A -85,B 0,C 180,E1 -4396.596,E2 -4396.596} C_VEL
LIN {X 0,Y 448.204,Z 993.409,A -85,B 0,C 180,E1 -4399.329,E2 -4399.329} C_VEL
LIN {X 0,Y 448.001,Z 998.814,A -85,B 0,C 180,E1 -4402.046,E2 -4402.046} C_VEL
LIN {X 0,Y 447.91,Z 1002.74,A -85,B 0,C 180,E1 -4404.877,E2 -4404.877} C_VEL
LIN {X 0,Y 447.901,Z 1004.832,A -85,B 0,C 180,E1 -4407.569,E2 -4407.569} C_VEL
LIN {X 0,Y 447.894,Z 1005.447,A -85,B 0,C 180,E1 -4410.511,E2 -4410.511} C_VEL
LIN {X 0,Y 447.904,Z 1004.418,A -85,B 0,C 180,E1 -4413.199,E2 -4413.199} C_VEL
LIN {X 0,Y 447.944,Z 1001.674,A -85,B 0,C 180,E1 -4416.022,E2 -4416.022} C_VEL
LIN {X 0,Y 448.052,Z 997.198,A -85,B 0,C 180,E1 -4418.857,E2 -4418.857} C_VEL
LIN {X 0,Y 448.301,Z 991.24,A -85,B 0,C 180,E1 -4421.579,E2 -4421.579} C_VEL
LIN {X 0,Y 448.774,Z 983.532,A -85,B 0,C 180,E1 -4424.318,E2 -4424.318} C_VEL
LIN {X 0,Y 449.56,Z 973.905,A -85,B 0,C 180,E1 -4427.072,E2 -4427.072} C_VEL
LIN {X 0,Y 450.683,Z 962.729,A -85,B 0,C 180,E1 -4429.707,E2 -4429.707} C_VEL
LIN {X 0,Y 451.741,Z 952.321,A -85,B 0,C 180,E1 -4431.692,E2 -4431.692} C_VEL
LIN {X 0,Y 453.329,Z 937.583,A -85,B 0,C 180,E1 -4434.081,E2 -4434.081} C_VEL
LIN {X 0,Y 455.228,Z 920.678,A -85,B 0,C 180,E1 -4436.408,E2 -4436.408} C_VEL
LIN {X 0,Y 457.304,Z 902.473,A -85,B 0,C 180,E1 -4438.537,E2 -4438.537} C_VEL
LIN {X 0,Y 459.573,Z 882.494,A -85,B 0,C 180,E1 -4440.51,E2 -4440.51} C_VEL
LIN {X 0,Y 461.773,Z 862.387,A -85,B 0,C 180,E1 -4442.185,E2 -4442.185} C_VEL
LIN {X 0,Y 463.917,Z 841.477,A -85,B 0,C 180,E1 -4443.635,E2 -4443.635} C_VEL
LIN {X 0,Y 465.951,Z 819.563,A -85,B 0,C 180,E1 -4444.88,E2 -4444.88} C_VEL
LIN {X 0,Y 467.732,Z 798.246,A -85,B 0,C 180,E1 -4445.854,E2 -4445.854} C_VEL
LIN {X 0,Y 469.242,Z 775.86,A -85,B 0,C 180,E1 -4446.632,E2 -4446.632} C_VEL
LIN {X 0,Y 470.464,Z 752.854,A -85,B 0,C 180,E1 -4447.197,E2 -4447.197} C_VEL
LIN {X 0,Y 471.639,Z 716.861,A -85,B 0,C 180,E1 -4447.814,E2 -4447.814} C_VEL
LIN {X 0,Y 476.837,Z 699.668,A -85,B 0,C 180,E1 -4448.595,E2 -4448.595} C_VEL
LIN {X 0,Y 483.646,Z 680.285,A -85,B 0,C 180,E1 -4449.395,E2 -4449.395} C_VEL
LIN {X 0,Y 491.126,Z 663.013,A -85,B 0,C 180,E1 -4449.964,E2 -4449.964} C_VEL
LIN {X 0,Y 497.694,Z 646.91,A -85,B 0,C 180,E1 -4450.534,E2 -4450.534} C_VEL
LIN {X 0,Y 507.544,Z 627.375,A -85,B 0,C 180,E1 -4451.071,E2 -4451.071} C_VEL
LIN {X 0,Y 523.17,Z 600.307,A -85,B 0,C 180,E1 -4451.608,E2 -4451.608} C_VEL
LIN {X 0,Y 532.837,Z 583.793,A -85,B 0,C 180,E1 -4451.885,E2 -4451.885} C_VEL
LIN {X 0,Y 521.501,Z 577.591,A -85,B 0,C 180,E1 -4453.234,E2 -4453.234} C_VEL
LIN {X 0,Y 510.965,Z 569.354,A -85,B 0,C 180,E1 -4454.739,E2 -4454.739} C_VEL
LIN {X 0,Y 502.648,Z 560.082,A -85,B 0,C 180,E1 -4456.225,E2 -4456.225} C_VEL
LIN {X 0,Y 496.477,Z 550.57,A -85,B 0,C 180,E1 -4457.573,E2 -4457.573} C_VEL
LIN {X 0,Y 490.834,Z 537.916,A -85,B 0,C 180,E1 -4459.164,E2 -4459.164} C_VEL
LIN {X 0,Y 487.08,Z 524.08,A -85,B 0,C 180,E1 -4460.704,E2 -4460.704} C_VEL
LIN {X 0,Y 484.992,Z 508.431,A -85,B 0,C 180,E1 -4462.245,E2 -4462.245} C_VEL
LIN {X 0,Y 484.626,Z 491.089,A -85,B 0,C 180,E1 -4463.774,E2 -4463.774} C_VEL
LIN {X 0,Y 486.337,Z 467.948,A -85,B 0,C 180,E1 -4465.572,E2 -4465.572} C_VEL
LIN {X 0,Y 488.621,Z 445.413,A -85,B 0,C 180,E1 -4467.302,E2 -4467.302} C_VEL
LIN {X 0,Y 478.715,Z 427.219,A -85,B 0,C 180,E1 -4470.468,E2 -4470.468} C_VEL
LIN {X 0,Y 471.126,Z 413.627,A -85,B 0,C 180,E1 -4473.044,E2 -4473.044} C_VEL
LIN {X 0,Y 463.483,Z 400.048,A -85,B 0,C 180,E1 -4475.803,E2 -4475.803} C_VEL
LIN {X 0,Y 459.594,Z 393.662,A -85,B 0,C 180,E1 -4477.217,E2 -4477.217} C_VEL
LIN {X 0,Y 457.503,Z 389.804,A -85,B 0,C 180,E1 -4478.055,E2 -4478.055} C_VEL
LIN {X 0,Y 455.15,Z 385.517,A -85,B 0,C 180,E1 -4479.006,E2 -4479.006} C_VEL
LIN {X 0,Y 452.545,Z 381.646,A -85,B 0,C 180,E1 -4479.974,E2 -4479.974} C_VEL
LIN {X 0,Y 451.809,Z 379.835,A -85,B 0,C 180,E1 -4480.344,E2 -4480.344} C_VEL
LIN {X 0,Y 449.813,Z 377.256,A -85,B 0,C 180,E1 -4481.063,E2 -4481.063} C_VEL
LIN {X 0,Y 449.101,Z 374.792,A -85,B 0,C 180,E1 -4481.571,E2 -4481.571} C_VEL
LIN {X 0,Y 449.139,Z 374.788,A -85,B 0,C 180,E1 -4485.167,E2 -4485.167} C_VEL
LIN {X 0,Y 449.11,Z 374.794,A -85,B 0,C 180,E1 -4488.962,E2 -4488.962} C_VEL
LIN {X 0,Y 449.135,Z 374.789,A -85,B 0,C 180,E1 -4492.582,E2 -4492.582} C_VEL
LIN {X 0,Y 449.116,Z 374.792,A -85,B 0,C 180,E1 -4496.426,E2 -4496.426} C_VEL
LIN {X 0,Y 449.121,Z 374.793,A -85,B 0,C 180,E1 -4500.128,E2 -4500.128} C_VEL
LIN {X 0,Y 449.093,Z 374.799,A -85,B 0,C 180,E1 -4503.958,E2 -4503.958} C_VEL
LIN {X 0,Y 449.138,Z 374.79,A -85,B 0,C 180,E1 -4507.676,E2 -4507.676} C_VEL
LIN {X 0,Y 449.127,Z 374.794,A -85,B 0,C 180,E1 -4511.428,E2 -4511.428} C_VEL
LIN {X 0,Y 449.122,Z 374.788,A -85,B 0,C 180,E1 -4515.098,E2 -4515.098} C_VEL
LIN {X 0,Y 449.1,Z 374.791,A -85,B 0,C 180,E1 -4518.88,E2 -4518.88} C_VEL
LIN {X 0,Y 449.139,Z 374.792,A -85,B 0,C 180,E1 -4522.514,E2 -4522.514} C_VEL
LIN {X 0,Y 449.103,Z 374.789,A -85,B 0,C 180,E1 -4526.299,E2 -4526.299} C_VEL
LIN {X 0,Y 449.139,Z 374.788,A -85,B 0,C 180,E1 -4529.912,E2 -4529.912} C_VEL
LIN {X 0,Y 449.112,Z 374.794,A -85,B 0,C 180,E1 -4533.666,E2 -4533.666} C_VEL
LIN {X 0,Y 449.123,Z 374.76,A -85,B 0,C 180,E1 -4537.367,E2 -4537.367} C_VEL
LIN {X 0,Y 449.088,Z 374.783,A -85,B 0,C 180,E1 -4541.056,E2 -4541.056} C_VEL
LIN {X 0,Y 449.136,Z 374.792,A -85,B 0,C 180,E1 -4544.753,E2 -4544.753} C_VEL
LIN {X 0,Y 449.125,Z 374.783,A -85,B 0,C 180,E1 -4548.439,E2 -4548.439} C_VEL
LIN {X 0,Y 449.132,Z 374.949,A -85,B 0,C 180,E1 -4549.804,E2 -4549.804} C_VEL
LIN {X 0,Y 450.393,Z 378.194,A -85,B 0,C 180,E1 -4550.185,E2 -4550.185} C_VEL
LIN {X 0,Y 457.851,Z 395.28,A -85,B 0,C 180,E1 -4552.305,E2 -4552.305} C_VEL
LIN {X 0,Y 465.63,Z 415.794,A -85,B 0,C 180,E1 -4554.716,E2 -4554.716} C_VEL
LIN {X 0,Y 463.649,Z 460.249,A -85,B 0,C 180,E1 -4558.175,E2 -4558.175} C_VEL
LIN {X 0,Y 463.061,Z 487.76,A -85,B 0,C 180,E1 -4560.139,E2 -4560.139} C_VEL
LIN {X 0,Y 464.166,Z 496.37,A -85,B 0,C 180,E1 -4560.372,E2 -4560.372} C_VEL
LIN {X 0,Y 463.286,Z 544.923,A -85,B 0,C 180,E1 -4561.164,E2 -4561.164} C_VEL
LIN {X 0,Y 462.29,Z 552.608,A -85,B 0,C 180,E1 -4561.229,E2 -4561.229} C_VEL
LIN {X 0,Y 456.49,Z 573.049,A -85,B 0,C 180,E1 -4561.176,E2 -4561.176} C_VEL
LIN {X 0,Y 455.728,Z 579.645,A -85,B 0,C 180,E1 -4561.239,E2 -4561.239} C_VEL
LIN {X 0,Y 453.765,Z 697.056,A -85,B 0,C 180,E1 -4563.214,E2 -4563.214} C_VEL
LIN {X 0,Y 453.3,Z 715.713,A -85,B 0,C 180,E1 -4563.753,E2 -4563.753} C_VEL
LIN {X 0,Y 452.558,Z 733.125,A -85,B 0,C 180,E1 -4564.481,E2 -4564.481} C_VEL
LIN {X 0,Y 451.495,Z 750.386,A -85,B 0,C 180,E1 -4565.435,E2 -4565.435} C_VEL
LIN {X 0,Y 450.252,Z 766.649,A -85,B 0,C 180,E1 -4566.578,E2 -4566.578} C_VEL
LIN {X 0,Y 448.875,Z 782.366,A -85,B 0,C 180,E1 -4567.949,E2 -4567.949} C_VEL
LIN {X 0,Y 447.382,Z 797.186,A -85,B 0,C 180,E1 -4569.527,E2 -4569.527} C_VEL
LIN {X 0,Y 445.918,Z 810.85,A -85,B 0,C 180,E1 -4571.299,E2 -4571.299} C_VEL
LIN {X 0,Y 444.527,Z 823.307,A -85,B 0,C 180,E1 -4573.268,E2 -4573.268} C_VEL
LIN {X 0,Y 443.332,Z 834.178,A -85,B 0,C 180,E1 -4575.369,E2 -4575.369} C_VEL
LIN {X 0,Y 442.378,Z 843.513,A -85,B 0,C 180,E1 -4577.601,E2 -4577.601} C_VEL
LIN {X 0,Y 441.633,Z 851.307,A -85,B 0,C 180,E1 -4579.961,E2 -4579.961} C_VEL
LIN {X 0,Y 441.14,Z 857.506,A -85,B 0,C 180,E1 -4582.446,E2 -4582.446} C_VEL
LIN {X 0,Y 440.874,Z 861.827,A -85,B 0,C 180,E1 -4584.926,E2 -4584.926} C_VEL
LIN {X 0,Y 440.728,Z 864.418,A -85,B 0,C 180,E1 -4587.4,E2 -4587.4} C_VEL
LIN {X 0,Y 440.686,Z 865.355,A -85,B 0,C 180,E1 -4589.87,E2 -4589.87} C_VEL
LIN {X 0,Y 440.726,Z 864.594,A -85,B 0,C 180,E1 -4592.471,E2 -4592.471} C_VEL
LIN {X 0,Y 440.865,Z 862.154,A -85,B 0,C 180,E1 -4594.944,E2 -4594.944} C_VEL
LIN {X 0,Y 441.116,Z 857.98,A -85,B 0,C 180,E1 -4597.424,E2 -4597.424} C_VEL
LIN {X 0,Y 441.549,Z 852.322,A -85,B 0,C 180,E1 -4599.778,E2 -4599.778} C_VEL
LIN {X 0,Y 442.204,Z 845.291,A -85,B 0,C 180,E1 -4602.007,E2 -4602.007} C_VEL
LIN {X 0,Y 443.1,Z 836.379,A -85,B 0,C 180,E1 -4604.239,E2 -4604.239} C_VEL
LIN {X 0,Y 444.222,Z 825.982,A -85,B 0,C 180,E1 -4606.341,E2 -4606.341} C_VEL
LIN {X 0,Y 445.575,Z 813.891,A -85,B 0,C 180,E1 -4608.34,E2 -4608.34} C_VEL
LIN {X 0,Y 447.016,Z 800.592,A -85,B 0,C 180,E1 -4610.149,E2 -4610.149} C_VEL
LIN {X 0,Y 448.458,Z 786.586,A -85,B 0,C 180,E1 -4611.723,E2 -4611.723} C_VEL
